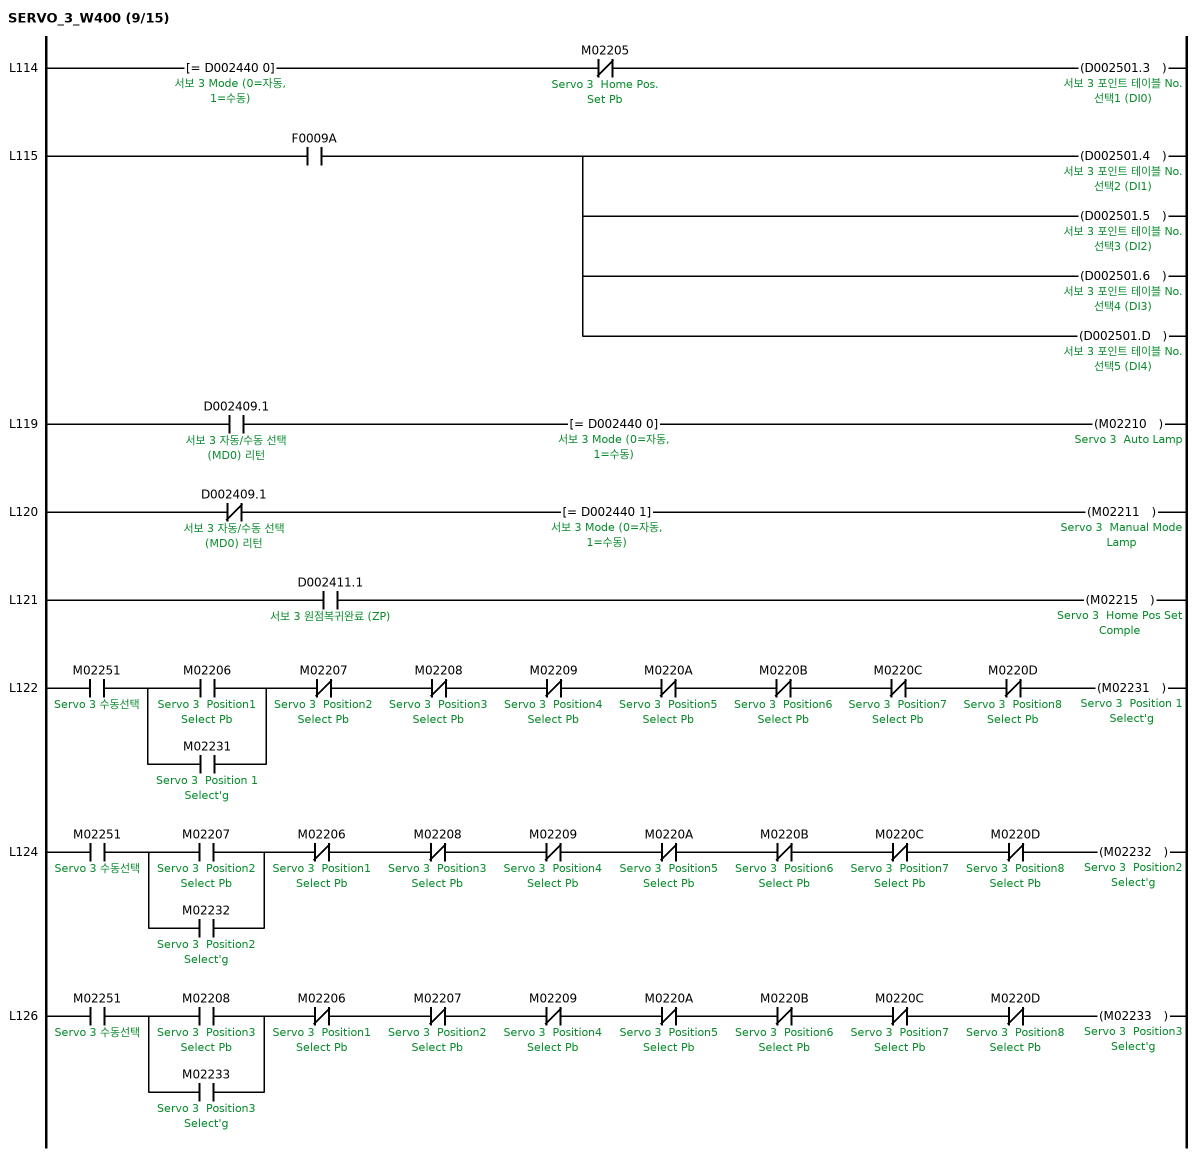
[picture p312: SERVO_3_W400 rungs L114-L126]
; L114
LOAD=     D002440 0	// 서보 3 Mode (0=자동, 1=수동)
AND NOT   M02205	// Servo 3  Home Pos. Set Pb
OUT       D002501.3	// 서보 3 포인트 테이블 No. 선택1 (DI0)
; L115
LOAD      F0009A
OUT       D002501.4	// 서보 3 포인트 테이블 No. 선택2 (DI1)
OUT       D002501.5	// 서보 3 포인트 테이블 No. 선택3 (DI2)
OUT       D002501.6	// 서보 3 포인트 테이블 No. 선택4 (DI3)
OUT       D002501.D	// 서보 3 포인트 테이블 No. 선택5 (DI4)
; L119
LOAD      D002409.1	// 서보 3 자동/수동 선택 (MD0) 리턴
AND=      D002440 0	// 서보 3 Mode (0=자동, 1=수동)
OUT       M02210	// Servo 3  Auto Lamp
; L120
LOAD NOT  D002409.1	// 서보 3 자동/수동 선택 (MD0) 리턴
AND=      D002440 1	// 서보 3 Mode (0=자동, 1=수동)
OUT       M02211	// Servo 3  Manual Mode Lamp
; L121
LOAD      D002411.1	// 서보 3 원점복귀완료 (ZP)
OUT       M02215	// Servo 3  Home Pos Set Comple
; L122
LOAD      M02251	// Servo 3 수동선택
LOAD      M02206	// Servo 3  Position1 Select Pb
OR        M02231	// Servo 3  Position 1 Select'g
AND LOAD
AND NOT   M02207	// Servo 3  Position2 Select Pb
AND NOT   M02208	// Servo 3  Position3 Select Pb
AND NOT   M02209	// Servo 3  Position4 Select Pb
AND NOT   M0220A	// Servo 3  Position5 Select Pb
AND NOT   M0220B	// Servo 3  Position6 Select Pb
AND NOT   M0220C	// Servo 3  Position7 Select Pb
AND NOT   M0220D	// Servo 3  Position8 Select Pb
OUT       M02231	// Servo 3  Position 1 Select'g
; L124
LOAD      M02251	// Servo 3 수동선택
LOAD      M02207	// Servo 3  Position2 Select Pb
OR        M02232	// Servo 3  Position2 Select'g
AND LOAD
AND NOT   M02206	// Servo 3  Position1 Select Pb
AND NOT   M02208	// Servo 3  Position3 Select Pb
AND NOT   M02209	// Servo 3  Position4 Select Pb
AND NOT   M0220A	// Servo 3  Position5 Select Pb
AND NOT   M0220B	// Servo 3  Position6 Select Pb
AND NOT   M0220C	// Servo 3  Position7 Select Pb
AND NOT   M0220D	// Servo 3  Position8 Select Pb
OUT       M02232	// Servo 3  Position2 Select'g
; L126
LOAD      M02251	// Servo 3 수동선택
LOAD      M02208	// Servo 3  Position3 Select Pb
OR        M02233	// Servo 3  Position3 Select'g
AND LOAD
AND NOT   M02206	// Servo 3  Position1 Select Pb
AND NOT   M02207	// Servo 3  Position2 Select Pb
AND NOT   M02209	// Servo 3  Position4 Select Pb
AND NOT   M0220A	// Servo 3  Position5 Select Pb
AND NOT   M0220B	// Servo 3  Position6 Select Pb
AND NOT   M0220C	// Servo 3  Position7 Select Pb
AND NOT   M0220D	// Servo 3  Position8 Select Pb
OUT       M02233	// Servo 3  Position3 Select'g

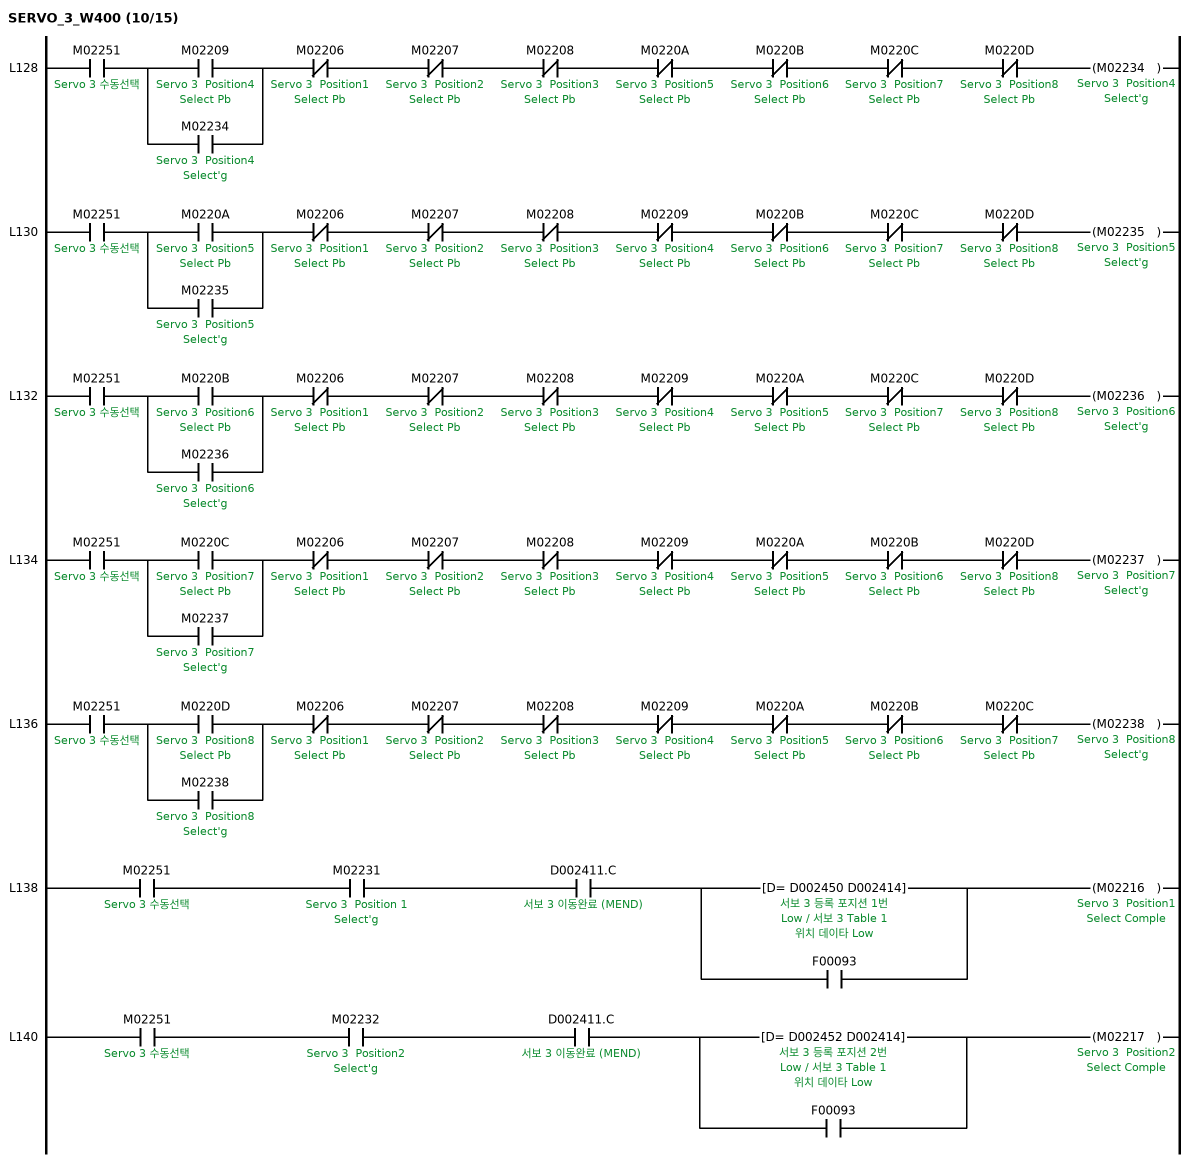
; L128
LOAD      M02251	// Servo 3 수동선택
LOAD      M02209	// Servo 3  Position4 Select Pb
OR        M02234	// Servo 3  Position4 Select'g
AND LOAD
AND NOT   M02206	// Servo 3  Position1 Select Pb
AND NOT   M02207	// Servo 3  Position2 Select Pb
AND NOT   M02208	// Servo 3  Position3 Select Pb
AND NOT   M0220A	// Servo 3  Position5 Select Pb
AND NOT   M0220B	// Servo 3  Position6 Select Pb
AND NOT   M0220C	// Servo 3  Position7 Select Pb
AND NOT   M0220D	// Servo 3  Position8 Select Pb
OUT       M02234	// Servo 3  Position4 Select'g
; L130
LOAD      M02251	// Servo 3 수동선택
LOAD      M0220A	// Servo 3  Position5 Select Pb
OR        M02235	// Servo 3  Position5 Select'g
AND LOAD
AND NOT   M02206	// Servo 3  Position1 Select Pb
AND NOT   M02207	// Servo 3  Position2 Select Pb
AND NOT   M02208	// Servo 3  Position3 Select Pb
AND NOT   M02209	// Servo 3  Position4 Select Pb
AND NOT   M0220B	// Servo 3  Position6 Select Pb
AND NOT   M0220C	// Servo 3  Position7 Select Pb
AND NOT   M0220D	// Servo 3  Position8 Select Pb
OUT       M02235	// Servo 3  Position5 Select'g
; L132
LOAD      M02251	// Servo 3 수동선택
LOAD      M0220B	// Servo 3  Position6 Select Pb
OR        M02236	// Servo 3  Position6 Select'g
AND LOAD
AND NOT   M02206	// Servo 3  Position1 Select Pb
AND NOT   M02207	// Servo 3  Position2 Select Pb
AND NOT   M02208	// Servo 3  Position3 Select Pb
AND NOT   M02209	// Servo 3  Position4 Select Pb
AND NOT   M0220A	// Servo 3  Position5 Select Pb
AND NOT   M0220C	// Servo 3  Position7 Select Pb
AND NOT   M0220D	// Servo 3  Position8 Select Pb
OUT       M02236	// Servo 3  Position6 Select'g
; L134
LOAD      M02251	// Servo 3 수동선택
LOAD      M0220C	// Servo 3  Position7 Select Pb
OR        M02237	// Servo 3  Position7 Select'g
AND LOAD
AND NOT   M02206	// Servo 3  Position1 Select Pb
AND NOT   M02207	// Servo 3  Position2 Select Pb
AND NOT   M02208	// Servo 3  Position3 Select Pb
AND NOT   M02209	// Servo 3  Position4 Select Pb
AND NOT   M0220A	// Servo 3  Position5 Select Pb
AND NOT   M0220B	// Servo 3  Position6 Select Pb
AND NOT   M0220D	// Servo 3  Position8 Select Pb
OUT       M02237	// Servo 3  Position7 Select'g
; L136
LOAD      M02251	// Servo 3 수동선택
LOAD      M0220D	// Servo 3  Position8 Select Pb
OR        M02238	// Servo 3  Position8 Select'g
AND LOAD
AND NOT   M02206	// Servo 3  Position1 Select Pb
AND NOT   M02207	// Servo 3  Position2 Select Pb
AND NOT   M02208	// Servo 3  Position3 Select Pb
AND NOT   M02209	// Servo 3  Position4 Select Pb
AND NOT   M0220A	// Servo 3  Position5 Select Pb
AND NOT   M0220B	// Servo 3  Position6 Select Pb
AND NOT   M0220C	// Servo 3  Position7 Select Pb
OUT       M02238	// Servo 3  Position8 Select'g
; L138
LOAD      M02251	// Servo 3 수동선택
AND       M02231	// Servo 3  Position 1 Select'g
AND       D002411.C	// 서보 3 이동완료 (MEND)
LOADD=    D002450 D002414	// 서보 3 등록 포지션 1번 Low / 서보 3 Table 1 위치 데이타 Low
OR        F00093
AND LOAD
OUT       M02216	// Servo 3  Position1 Select Comple
; L140
LOAD      M02251	// Servo 3 수동선택
AND       M02232	// Servo 3  Position2 Select'g
AND       D002411.C	// 서보 3 이동완료 (MEND)
LOADD=    D002452 D002414	// 서보 3 등록 포지션 2번 Low / 서보 3 Table 1 위치 데이타 Low
OR        F00093
AND LOAD
OUT       M02217	// Servo 3  Position2 Select Comple

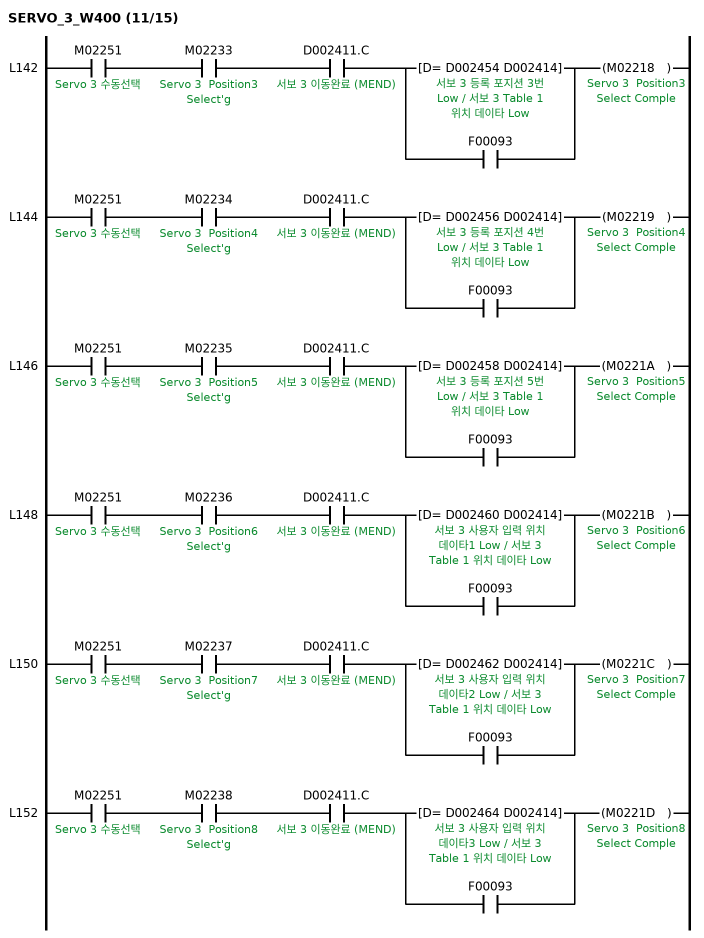
; L142
LOAD      M02251	// Servo 3 수동선택
AND       M02233	// Servo 3  Position3 Select'g
AND       D002411.C	// 서보 3 이동완료 (MEND)
LOADD=    D002454 D002414	// 서보 3 등록 포지션 3번 Low / 서보 3 Table 1 위치 데이타 Low
OR        F00093
AND LOAD
OUT       M02218	// Servo 3  Position3 Select Comple
; L144
LOAD      M02251	// Servo 3 수동선택
AND       M02234	// Servo 3  Position4 Select'g
AND       D002411.C	// 서보 3 이동완료 (MEND)
LOADD=    D002456 D002414	// 서보 3 등록 포지션 4번 Low / 서보 3 Table 1 위치 데이타 Low
OR        F00093
AND LOAD
OUT       M02219	// Servo 3  Position4 Select Comple
; L146
LOAD      M02251	// Servo 3 수동선택
AND       M02235	// Servo 3  Position5 Select'g
AND       D002411.C	// 서보 3 이동완료 (MEND)
LOADD=    D002458 D002414	// 서보 3 등록 포지션 5번 Low / 서보 3 Table 1 위치 데이타 Low
OR        F00093
AND LOAD
OUT       M0221A	// Servo 3  Position5 Select Comple
; L148
LOAD      M02251	// Servo 3 수동선택
AND       M02236	// Servo 3  Position6 Select'g
AND       D002411.C	// 서보 3 이동완료 (MEND)
LOADD=    D002460 D002414	// 서보 3 사용자 입력 위치 데이타1 Low / 서보 3 Table 1 위치 데이타 Low
OR        F00093
AND LOAD
OUT       M0221B	// Servo 3  Position6 Select Comple
; L150
LOAD      M02251	// Servo 3 수동선택
AND       M02237	// Servo 3  Position7 Select'g
AND       D002411.C	// 서보 3 이동완료 (MEND)
LOADD=    D002462 D002414	// 서보 3 사용자 입력 위치 데이타2 Low / 서보 3 Table 1 위치 데이타 Low
OR        F00093
AND LOAD
OUT       M0221C	// Servo 3  Position7 Select Comple
; L152
LOAD      M02251	// Servo 3 수동선택
AND       M02238	// Servo 3  Position8 Select'g
AND       D002411.C	// 서보 3 이동완료 (MEND)
LOADD=    D002464 D002414	// 서보 3 사용자 입력 위치 데이타3 Low / 서보 3 Table 1 위치 데이타 Low
OR        F00093
AND LOAD
OUT       M0221D	// Servo 3  Position8 Select Comple

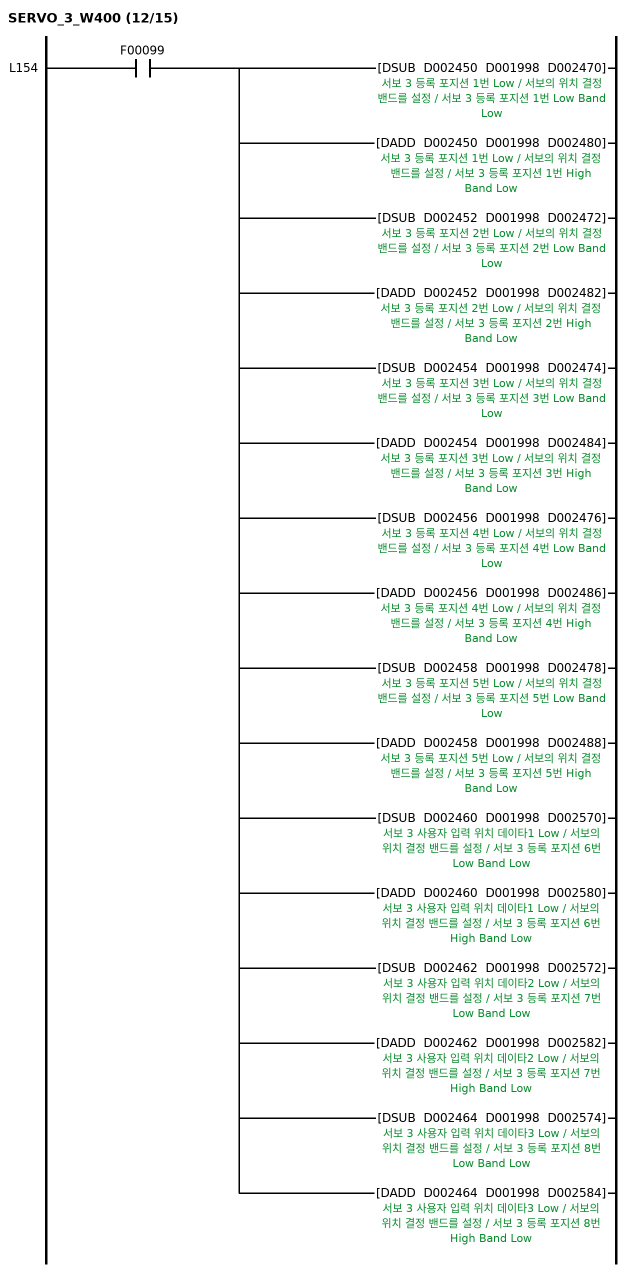
; L154
LOAD      F00099
DSUB      D002450 D001998 D002470	// 서보 3 등록 포지션 1번 Low / 서보의 위치 결정 밴드를 설정 / 서보 3 등록 포지션 1번 Low Band Low
DADD      D002450 D001998 D002480	// 서보 3 등록 포지션 1번 Low / 서보의 위치 결정 밴드를 설정 / 서보 3 등록 포지션 1번 High Band Low
DSUB      D002452 D001998 D002472	// 서보 3 등록 포지션 2번 Low / 서보의 위치 결정 밴드를 설정 / 서보 3 등록 포지션 2번 Low Band Low
DADD      D002452 D001998 D002482	// 서보 3 등록 포지션 2번 Low / 서보의 위치 결정 밴드를 설정 / 서보 3 등록 포지션 2번 High Band Low
DSUB      D002454 D001998 D002474	// 서보 3 등록 포지션 3번 Low / 서보의 위치 결정 밴드를 설정 / 서보 3 등록 포지션 3번 Low Band Low
DADD      D002454 D001998 D002484	// 서보 3 등록 포지션 3번 Low / 서보의 위치 결정 밴드를 설정 / 서보 3 등록 포지션 3번 High Band Low
DSUB      D002456 D001998 D002476	// 서보 3 등록 포지션 4번 Low / 서보의 위치 결정 밴드를 설정 / 서보 3 등록 포지션 4번 Low Band Low
DADD      D002456 D001998 D002486	// 서보 3 등록 포지션 4번 Low / 서보의 위치 결정 밴드를 설정 / 서보 3 등록 포지션 4번 High Band Low
DSUB      D002458 D001998 D002478	// 서보 3 등록 포지션 5번 Low / 서보의 위치 결정 밴드를 설정 / 서보 3 등록 포지션 5번 Low Band Low
DADD      D002458 D001998 D002488	// 서보 3 등록 포지션 5번 Low / 서보의 위치 결정 밴드를 설정 / 서보 3 등록 포지션 5번 High Band Low
DSUB      D002460 D001998 D002570	// 서보 3 사용자 입력 위치 데이타1 Low / 서보의 위치 결정 밴드를 설정 / 서보 3 등록 포지션 6번 Low Band Low
DADD      D002460 D001998 D002580	// 서보 3 사용자 입력 위치 데이타1 Low / 서보의 위치 결정 밴드를 설정 / 서보 3 등록 포지션 6번 High Band Low
DSUB      D002462 D001998 D002572	// 서보 3 사용자 입력 위치 데이타2 Low / 서보의 위치 결정 밴드를 설정 / 서보 3 등록 포지션 7번 Low Band Low
DADD      D002462 D001998 D002582	// 서보 3 사용자 입력 위치 데이타2 Low / 서보의 위치 결정 밴드를 설정 / 서보 3 등록 포지션 7번 High Band Low
DSUB      D002464 D001998 D002574	// 서보 3 사용자 입력 위치 데이타3 Low / 서보의 위치 결정 밴드를 설정 / 서보 3 등록 포지션 8번 Low Band Low
DADD      D002464 D001998 D002584	// 서보 3 사용자 입력 위치 데이타3 Low / 서보의 위치 결정 밴드를 설정 / 서보 3 등록 포지션 8번 High Band Low

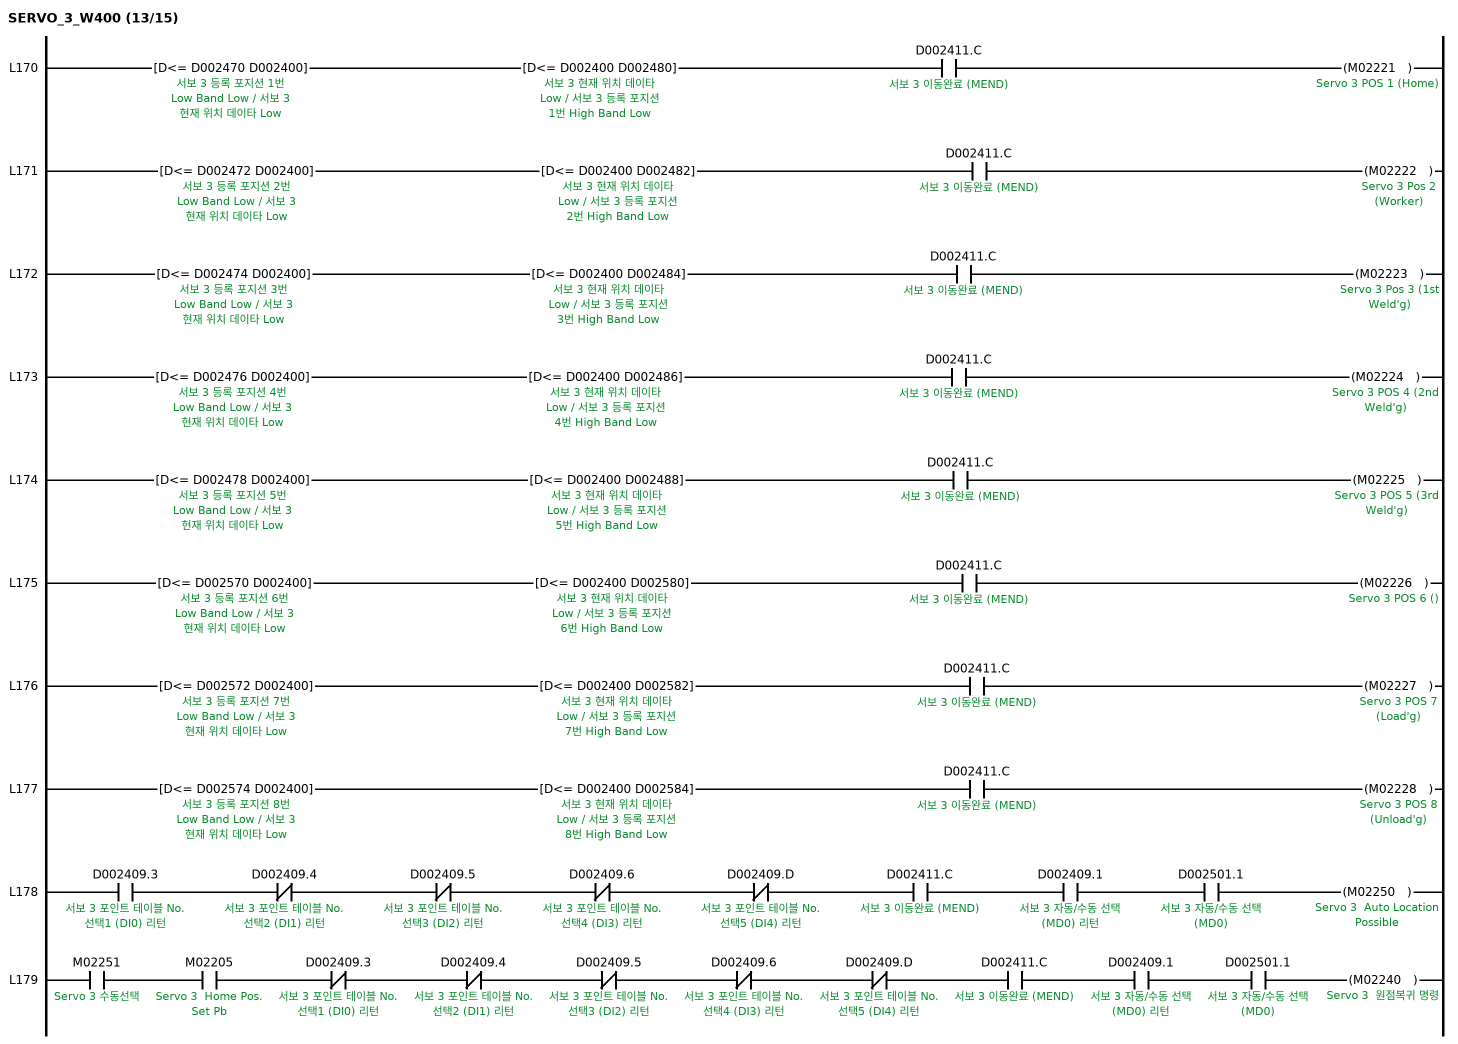
; L170
LOADD<=   D002470 D002400	// 서보 3 등록 포지션 1번 Low Band Low / 서보 3 현재 위치 데이타 Low
ANDD<=    D002400 D002480	// 서보 3 현재 위치 데이타 Low / 서보 3 등록 포지션 1번 High Band Low
AND       D002411.C	// 서보 3 이동완료 (MEND)
OUT       M02221	// Servo 3 POS 1 (Home)
; L171
LOADD<=   D002472 D002400	// 서보 3 등록 포지션 2번 Low Band Low / 서보 3 현재 위치 데이타 Low
ANDD<=    D002400 D002482	// 서보 3 현재 위치 데이타 Low / 서보 3 등록 포지션 2번 High Band Low
AND       D002411.C	// 서보 3 이동완료 (MEND)
OUT       M02222	// Servo 3 Pos 2 (Worker)
; L172
LOADD<=   D002474 D002400	// 서보 3 등록 포지션 3번 Low Band Low / 서보 3 현재 위치 데이타 Low
ANDD<=    D002400 D002484	// 서보 3 현재 위치 데이타 Low / 서보 3 등록 포지션 3번 High Band Low
AND       D002411.C	// 서보 3 이동완료 (MEND)
OUT       M02223	// Servo 3 Pos 3 (1st Weld'g)
; L173
LOADD<=   D002476 D002400	// 서보 3 등록 포지션 4번 Low Band Low / 서보 3 현재 위치 데이타 Low
ANDD<=    D002400 D002486	// 서보 3 현재 위치 데이타 Low / 서보 3 등록 포지션 4번 High Band Low
AND       D002411.C	// 서보 3 이동완료 (MEND)
OUT       M02224	// Servo 3 POS 4 (2nd Weld'g)
; L174
LOADD<=   D002478 D002400	// 서보 3 등록 포지션 5번 Low Band Low / 서보 3 현재 위치 데이타 Low
ANDD<=    D002400 D002488	// 서보 3 현재 위치 데이타 Low / 서보 3 등록 포지션 5번 High Band Low
AND       D002411.C	// 서보 3 이동완료 (MEND)
OUT       M02225	// Servo 3 POS 5 (3rd Weld'g)
; L175
LOADD<=   D002570 D002400	// 서보 3 등록 포지션 6번 Low Band Low / 서보 3 현재 위치 데이타 Low
ANDD<=    D002400 D002580	// 서보 3 현재 위치 데이타 Low / 서보 3 등록 포지션 6번 High Band Low
AND       D002411.C	// 서보 3 이동완료 (MEND)
OUT       M02226	// Servo 3 POS 6 ()
; L176
LOADD<=   D002572 D002400	// 서보 3 등록 포지션 7번 Low Band Low / 서보 3 현재 위치 데이타 Low
ANDD<=    D002400 D002582	// 서보 3 현재 위치 데이타 Low / 서보 3 등록 포지션 7번 High Band Low
AND       D002411.C	// 서보 3 이동완료 (MEND)
OUT       M02227	// Servo 3 POS 7 (Load'g)
; L177
LOADD<=   D002574 D002400	// 서보 3 등록 포지션 8번 Low Band Low / 서보 3 현재 위치 데이타 Low
ANDD<=    D002400 D002584	// 서보 3 현재 위치 데이타 Low / 서보 3 등록 포지션 8번 High Band Low
AND       D002411.C	// 서보 3 이동완료 (MEND)
OUT       M02228	// Servo 3 POS 8 (Unload'g)
; L178
LOAD      D002409.3	// 서보 3 포인트 테이블 No. 선택1 (DI0) 리턴
AND NOT   D002409.4	// 서보 3 포인트 테이블 No. 선택2 (DI1) 리턴
AND NOT   D002409.5	// 서보 3 포인트 테이블 No. 선택3 (DI2) 리턴
AND NOT   D002409.6	// 서보 3 포인트 테이블 No. 선택4 (DI3) 리턴
AND NOT   D002409.D	// 서보 3 포인트 테이블 No. 선택5 (DI4) 리턴
AND       D002411.C	// 서보 3 이동완료 (MEND)
AND       D002409.1	// 서보 3 자동/수동 선택 (MD0) 리턴
AND       D002501.1	// 서보 3 자동/수동 선택 (MD0)
OUT       M02250	// Servo 3  Auto Location Possible
; L179
LOAD      M02251	// Servo 3 수동선택
AND       M02205	// Servo 3  Home Pos. Set Pb
AND NOT   D002409.3	// 서보 3 포인트 테이블 No. 선택1 (DI0) 리턴
AND NOT   D002409.4	// 서보 3 포인트 테이블 No. 선택2 (DI1) 리턴
AND NOT   D002409.5	// 서보 3 포인트 테이블 No. 선택3 (DI2) 리턴
AND NOT   D002409.6	// 서보 3 포인트 테이블 No. 선택4 (DI3) 리턴
AND NOT   D002409.D	// 서보 3 포인트 테이블 No. 선택5 (DI4) 리턴
AND       D002411.C	// 서보 3 이동완료 (MEND)
AND       D002409.1	// 서보 3 자동/수동 선택 (MD0) 리턴
AND       D002501.1	// 서보 3 자동/수동 선택 (MD0)
OUT       M02240	// Servo 3  원점복귀 명령

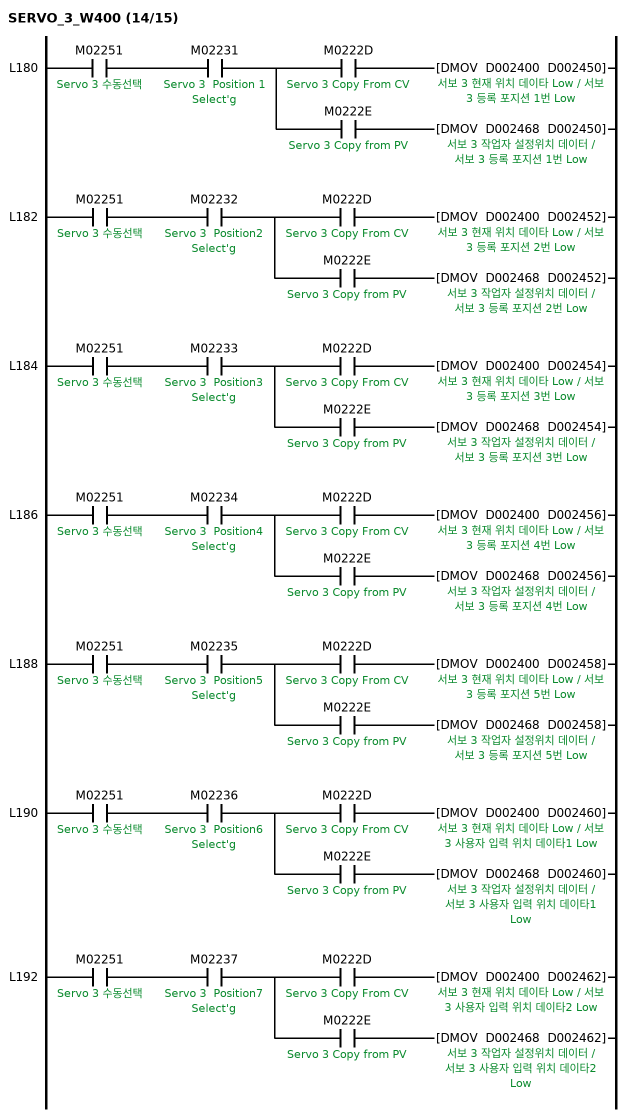
; L180
LOAD      M02251	// Servo 3 수동선택
AND       M02231	// Servo 3  Position 1 Select'g
MPUSH
AND       M0222D	// Servo 3 Copy From CV
DMOV      D002400 D002450	// 서보 3 현재 위치 데이타 Low / 서보 3 등록 포지션 1번 Low
MPOP
AND       M0222E	// Servo 3 Copy from PV
DMOV      D002468 D002450	// 서보 3 작업자 설정위치 데이터 / 서보 3 등록 포지션 1번 Low
; L182
LOAD      M02251	// Servo 3 수동선택
AND       M02232	// Servo 3  Position2 Select'g
MPUSH
AND       M0222D	// Servo 3 Copy From CV
DMOV      D002400 D002452	// 서보 3 현재 위치 데이타 Low / 서보 3 등록 포지션 2번 Low
MPOP
AND       M0222E	// Servo 3 Copy from PV
DMOV      D002468 D002452	// 서보 3 작업자 설정위치 데이터 / 서보 3 등록 포지션 2번 Low
; L184
LOAD      M02251	// Servo 3 수동선택
AND       M02233	// Servo 3  Position3 Select'g
MPUSH
AND       M0222D	// Servo 3 Copy From CV
DMOV      D002400 D002454	// 서보 3 현재 위치 데이타 Low / 서보 3 등록 포지션 3번 Low
MPOP
AND       M0222E	// Servo 3 Copy from PV
DMOV      D002468 D002454	// 서보 3 작업자 설정위치 데이터 / 서보 3 등록 포지션 3번 Low
; L186
LOAD      M02251	// Servo 3 수동선택
AND       M02234	// Servo 3  Position4 Select'g
MPUSH
AND       M0222D	// Servo 3 Copy From CV
DMOV      D002400 D002456	// 서보 3 현재 위치 데이타 Low / 서보 3 등록 포지션 4번 Low
MPOP
AND       M0222E	// Servo 3 Copy from PV
DMOV      D002468 D002456	// 서보 3 작업자 설정위치 데이터 / 서보 3 등록 포지션 4번 Low
; L188
LOAD      M02251	// Servo 3 수동선택
AND       M02235	// Servo 3  Position5 Select'g
MPUSH
AND       M0222D	// Servo 3 Copy From CV
DMOV      D002400 D002458	// 서보 3 현재 위치 데이타 Low / 서보 3 등록 포지션 5번 Low
MPOP
AND       M0222E	// Servo 3 Copy from PV
DMOV      D002468 D002458	// 서보 3 작업자 설정위치 데이터 / 서보 3 등록 포지션 5번 Low
; L190
LOAD      M02251	// Servo 3 수동선택
AND       M02236	// Servo 3  Position6 Select'g
MPUSH
AND       M0222D	// Servo 3 Copy From CV
DMOV      D002400 D002460	// 서보 3 현재 위치 데이타 Low / 서보 3 사용자 입력 위치 데이타1 Low
MPOP
AND       M0222E	// Servo 3 Copy from PV
DMOV      D002468 D002460	// 서보 3 작업자 설정위치 데이터 / 서보 3 사용자 입력 위치 데이타1 Low
; L192
LOAD      M02251	// Servo 3 수동선택
AND       M02237	// Servo 3  Position7 Select'g
MPUSH
AND       M0222D	// Servo 3 Copy From CV
DMOV      D002400 D002462	// 서보 3 현재 위치 데이타 Low / 서보 3 사용자 입력 위치 데이타2 Low
MPOP
AND       M0222E	// Servo 3 Copy from PV
DMOV      D002468 D002462	// 서보 3 작업자 설정위치 데이터 / 서보 3 사용자 입력 위치 데이타2 Low

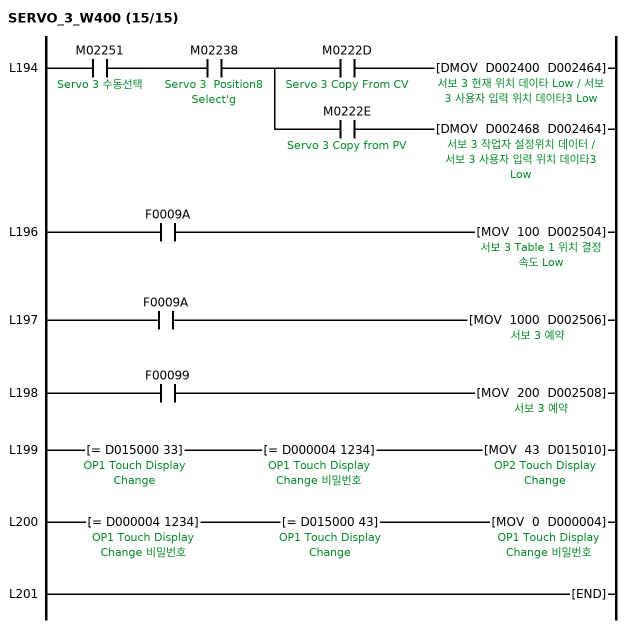
; L194
LOAD      M02251	// Servo 3 수동선택
AND       M02238	// Servo 3  Position8 Select'g
MPUSH
AND       M0222D	// Servo 3 Copy From CV
DMOV      D002400 D002464	// 서보 3 현재 위치 데이타 Low / 서보 3 사용자 입력 위치 데이타3 Low
MPOP
AND       M0222E	// Servo 3 Copy from PV
DMOV      D002468 D002464	// 서보 3 작업자 설정위치 데이터 / 서보 3 사용자 입력 위치 데이타3 Low
; L196
LOAD      F0009A
MOV       100 D002504	// 서보 3 Table 1 위치 결정 속도 Low
; L197
LOAD      F0009A
MOV       1000 D002506	// 서보 3 예약
; L198
LOAD      F00099
MOV       200 D002508	// 서보 3 예약
; L199
LOAD=     D015000 33	// OP1 Touch Display Change
AND=      D000004 1234	// OP1 Touch Display Change 비밀번호
MOV       43 D015010	// OP2 Touch Display Change
; L200
LOAD=     D000004 1234	// OP1 Touch Display Change 비밀번호
AND=      D015000 43	// OP1 Touch Display Change
MOV       0 D000004	// OP1 Touch Display Change 비밀번호
; L201
END

PROGRAM Robot_01_ARC (task: 스캔 프로그램)

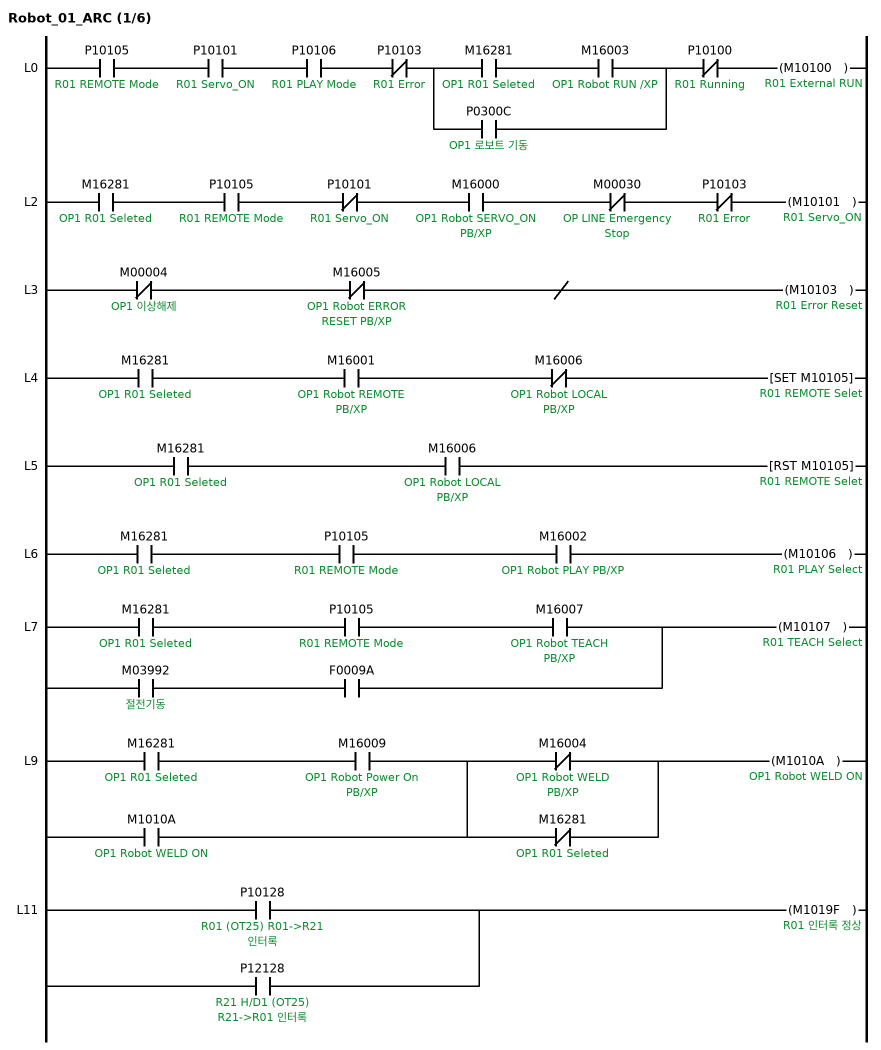
; L0
LOAD      P10105	// R01 REMOTE Mode
AND       P10101	// R01 Servo_ON
AND       P10106	// R01 PLAY Mode
AND NOT   P10103	// R01 Error
LOAD      M16281	// OP1 R01 Seleted
AND       M16003	// OP1 Robot RUN /XP
OR        P0300C	// OP1 로보트 기동
AND LOAD
AND NOT   P10100	// R01 Running
OUT       M10100	// R01 External RUN
; L2
LOAD      M16281	// OP1 R01 Seleted
AND       P10105	// R01 REMOTE Mode
AND NOT   P10101	// R01 Servo_ON
AND       M16000	// OP1 Robot SERVO_ON PB/XP
AND NOT   M00030	// OP LINE Emergency Stop
AND NOT   P10103	// R01 Error
OUT       M10101	// R01 Servo_ON
; L3
LOAD NOT  M00004	// OP1 이상해제
AND NOT   M16005	// OP1 Robot ERROR RESET PB/XP
NOT
OUT       M10103	// R01 Error Reset
; L4
LOAD      M16281	// OP1 R01 Seleted
AND       M16001	// OP1 Robot REMOTE PB/XP
AND NOT   M16006	// OP1 Robot LOCAL PB/XP
SET       M10105	// R01 REMOTE Selet
; L5
LOAD      M16281	// OP1 R01 Seleted
AND       M16006	// OP1 Robot LOCAL PB/XP
RST       M10105	// R01 REMOTE Selet
; L6
LOAD      M16281	// OP1 R01 Seleted
AND       P10105	// R01 REMOTE Mode
AND       M16002	// OP1 Robot PLAY PB/XP
OUT       M10106	// R01 PLAY Select
; L7
LOAD      M16281	// OP1 R01 Seleted
AND       P10105	// R01 REMOTE Mode
AND       M16007	// OP1 Robot TEACH PB/XP
LOAD      M03992	// 절전기동
AND       F0009A
OR LOAD
OUT       M10107	// R01 TEACH Select
; L9
LOAD      M16281	// OP1 R01 Seleted
AND       M16009	// OP1 Robot Power On PB/XP
OR        M1010A	// OP1 Robot WELD ON
LOAD NOT  M16004	// OP1 Robot WELD PB/XP
OR NOT    M16281	// OP1 R01 Seleted
AND LOAD
OUT       M1010A	// OP1 Robot WELD ON
; L11
LOAD      P10128	// R01 (OT25) R01->R21 인터록
OR        P12128	// R21 H/D1 (OT25) R21->R01 인터록
OUT       M1019F	// R01 인터록 정상

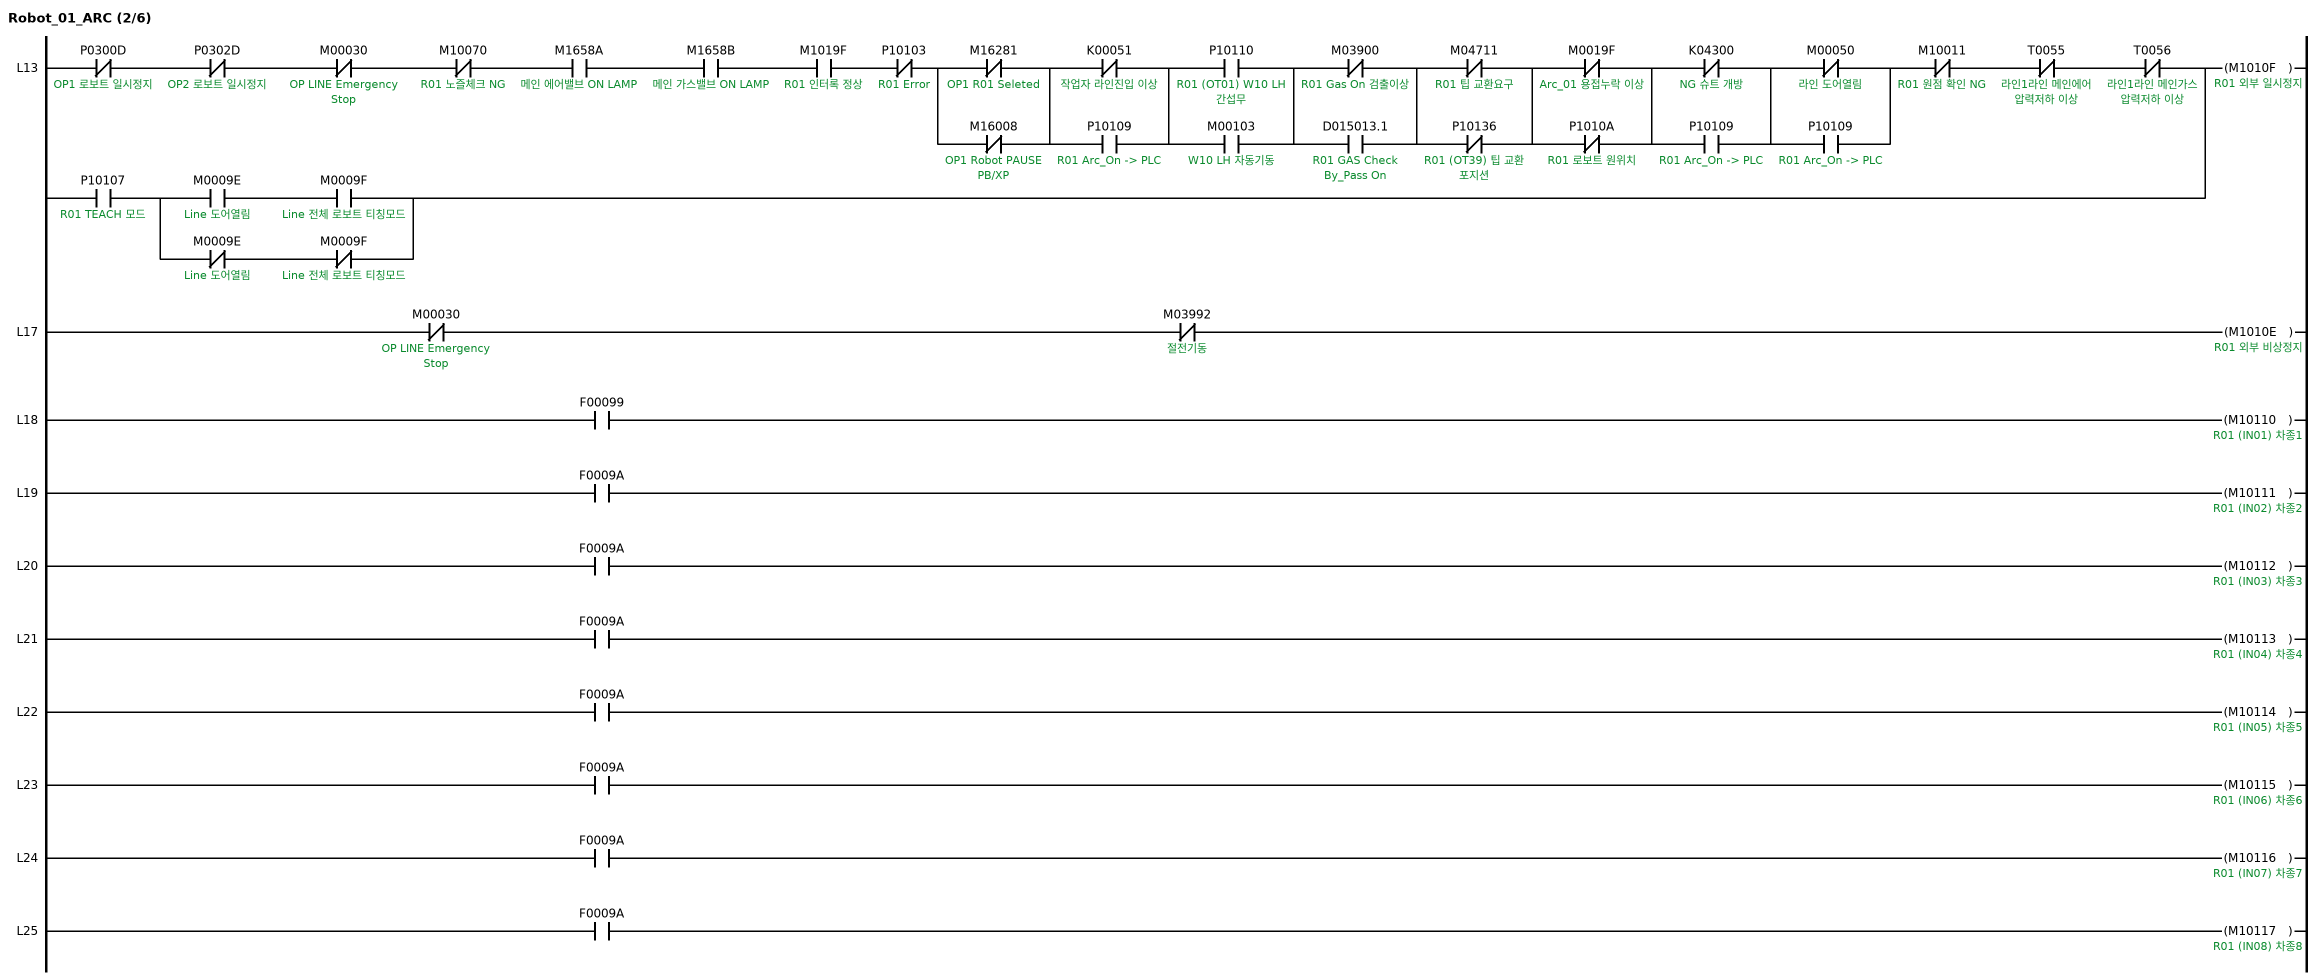
; L13
LOAD NOT  P0300D	// OP1 로보트 일시정지
AND NOT   P0302D	// OP2 로보트 일시정지
AND NOT   M00030	// OP LINE Emergency Stop
AND NOT   M10070	// R01 노즐체크 NG
AND       M1658A	// 메인 에어밸브 ON LAMP
AND       M1658B	// 메인 가스밸브 ON LAMP
AND       M1019F	// R01 인터록 정상
AND NOT   P10103	// R01 Error
LOAD NOT  M16281	// OP1 R01 Seleted
OR NOT    M16008	// OP1 Robot PAUSE PB/XP
AND LOAD
LOAD NOT  K00051	//  작업자 라인진입 이상
OR        P10109	// R01 Arc_On -> PLC
AND LOAD
LOAD      P10110	// R01 (OT01) W10 LH 간섭무
OR        M00103	// W10 LH 자동기동
AND LOAD
LOAD NOT  M03900	// R01 Gas On 검출이상
OR        D015013.1	// R01 GAS Check By_Pass On
AND LOAD
LOAD NOT  M04711	// R01 팁 교환요구
OR NOT    P10136	// R01 (OT39) 팁 교환 포지션
AND LOAD
LOAD NOT  M0019F	// Arc_01 용접누락 이상
OR NOT    P1010A	// R01 로보트 원위치
AND LOAD
LOAD NOT  K04300	// NG 슈트 개방
OR        P10109	// R01 Arc_On -> PLC
AND LOAD
LOAD NOT  M00050	// 라인 도어열림
OR        P10109	// R01 Arc_On -> PLC
AND LOAD
AND NOT   M10011	// R01 원점 확인 NG
AND NOT   T0055	// 라인1라인 메인에어 압력저하 이상
AND NOT   T0056	// 라인1라인 메인가스 압력저하 이상
LOAD      P10107	// R01 TEACH 모드
LOAD      M0009E	// Line 도어열림
AND       M0009F	// Line 전체 로보트 티칭모드
LOAD NOT  M0009E	// Line 도어열림
AND NOT   M0009F	// Line 전체 로보트 티칭모드
OR LOAD
AND LOAD
OR LOAD
OUT       M1010F	// R01 외부 일시정지
; L17
LOAD NOT  M00030	// OP LINE Emergency Stop
AND NOT   M03992	// 절전기동
OUT       M1010E	// R01 외부 비상정지 
; L18
LOAD      F00099
OUT       M10110	// R01 (IN01) 차종1
; L19
LOAD      F0009A
OUT       M10111	// R01 (IN02) 차종2
; L20
LOAD      F0009A
OUT       M10112	// R01 (IN03) 차종3
; L21
LOAD      F0009A
OUT       M10113	// R01 (IN04) 차종4
; L22
LOAD      F0009A
OUT       M10114	// R01 (IN05) 차종5
; L23
LOAD      F0009A
OUT       M10115	// R01 (IN06) 차종6
; L24
LOAD      F0009A
OUT       M10116	// R01 (IN07) 차종7
; L25
LOAD      F0009A
OUT       M10117	// R01 (IN08) 차종8

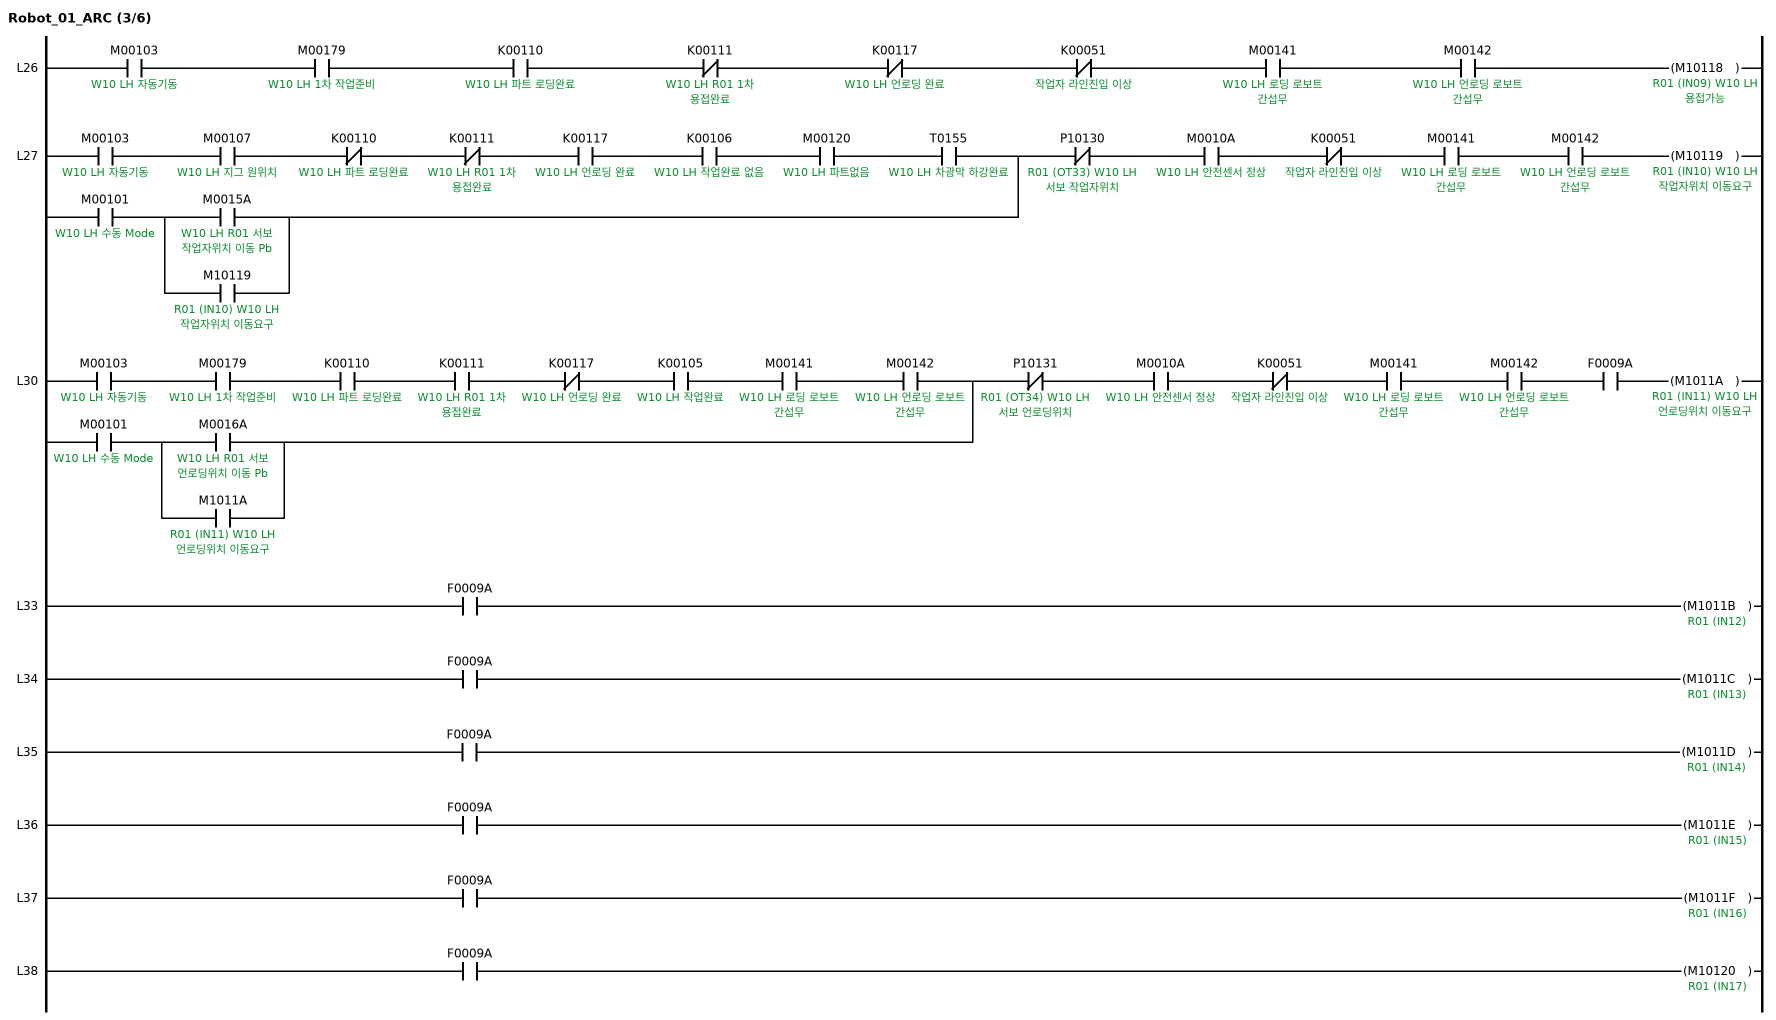
; L26
LOAD      M00103	// W10 LH 자동기동
AND       M00179	// W10 LH 1차 작업준비
AND       K00110	// W10 LH 파트 로딩완료
AND NOT   K00111	// W10 LH R01 1차 용접완료
AND NOT   K00117	// W10 LH 언로딩 완료
AND NOT   K00051	//  작업자 라인진입 이상
AND       M00141	// W10 LH 로딩 로보트 간섭무
AND       M00142	// W10 LH 언로딩 로보트 간섭무
OUT       M10118	// R01 (IN09) W10 LH 용접가능
; L27
LOAD      M00103	// W10 LH 자동기동
AND       M00107	// W10 LH 지그 원위치
AND NOT   K00110	// W10 LH 파트 로딩완료
AND NOT   K00111	// W10 LH R01 1차 용접완료
AND       K00117	// W10 LH 언로딩 완료
AND       K00106	// W10 LH 작업완료 없음
AND       M00120	// W10 LH 파트없음
AND       T0155	// W10 LH 차광막 하강완료
LOAD      M00101	// W10 LH 수동 Mode
LOAD      M0015A	// W10 LH R01 서보 작업자위치 이동 Pb
OR        M10119	// R01 (IN10) W10 LH 작업자위치 이동요구
AND LOAD
OR LOAD
AND NOT   P10130	// R01 (OT33) W10 LH 서보 작업자위치
AND       M0010A	// W10 LH 안전센서 정상
AND NOT   K00051	//  작업자 라인진입 이상
AND       M00141	// W10 LH 로딩 로보트 간섭무
AND       M00142	// W10 LH 언로딩 로보트 간섭무
OUT       M10119	// R01 (IN10) W10 LH 작업자위치 이동요구
; L30
LOAD      M00103	// W10 LH 자동기동
AND       M00179	// W10 LH 1차 작업준비
AND       K00110	// W10 LH 파트 로딩완료
AND       K00111	// W10 LH R01 1차 용접완료
AND NOT   K00117	// W10 LH 언로딩 완료
AND       K00105	// W10 LH 작업완료
AND       M00141	// W10 LH 로딩 로보트 간섭무
AND       M00142	// W10 LH 언로딩 로보트 간섭무
LOAD      M00101	// W10 LH 수동 Mode
LOAD      M0016A	// W10 LH R01 서보 언로딩위치 이동 Pb
OR        M1011A	// R01 (IN11) W10 LH 언로딩위치 이동요구
AND LOAD
OR LOAD
AND NOT   P10131	// R01 (OT34) W10 LH 서보 언로딩위치
AND       M0010A	// W10 LH 안전센서 정상
AND NOT   K00051	//  작업자 라인진입 이상
AND       M00141	// W10 LH 로딩 로보트 간섭무
AND       M00142	// W10 LH 언로딩 로보트 간섭무
AND       F0009A
OUT       M1011A	// R01 (IN11) W10 LH 언로딩위치 이동요구
; L33
LOAD      F0009A
OUT       M1011B	// R01 (IN12)
; L34
LOAD      F0009A
OUT       M1011C	// R01 (IN13)
; L35
LOAD      F0009A
OUT       M1011D	// R01 (IN14)
; L36
LOAD      F0009A
OUT       M1011E	// R01 (IN15)
; L37
LOAD      F0009A
OUT       M1011F	// R01 (IN16)
; L38
LOAD      F0009A
OUT       M10120	// R01 (IN17)

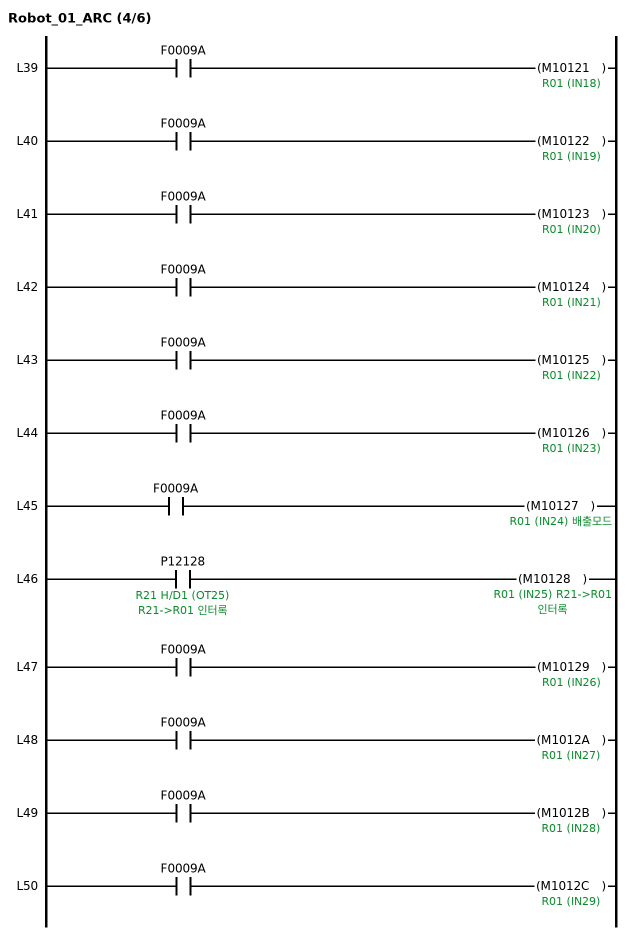
; L39
LOAD      F0009A
OUT       M10121	// R01 (IN18)
; L40
LOAD      F0009A
OUT       M10122	// R01 (IN19)
; L41
LOAD      F0009A
OUT       M10123	// R01 (IN20)
; L42
LOAD      F0009A
OUT       M10124	// R01 (IN21)
; L43
LOAD      F0009A
OUT       M10125	// R01 (IN22)
; L44
LOAD      F0009A
OUT       M10126	// R01 (IN23)
; L45
LOAD      F0009A
OUT       M10127	// R01 (IN24) 배출모드
; L46
LOAD      P12128	// R21 H/D1 (OT25) R21->R01 인터록
OUT       M10128	// R01 (IN25) R21->R01 인터록
; L47
LOAD      F0009A
OUT       M10129	// R01 (IN26)
; L48
LOAD      F0009A
OUT       M1012A	// R01 (IN27)
; L49
LOAD      F0009A
OUT       M1012B	// R01 (IN28)
; L50
LOAD      F0009A
OUT       M1012C	// R01 (IN29)

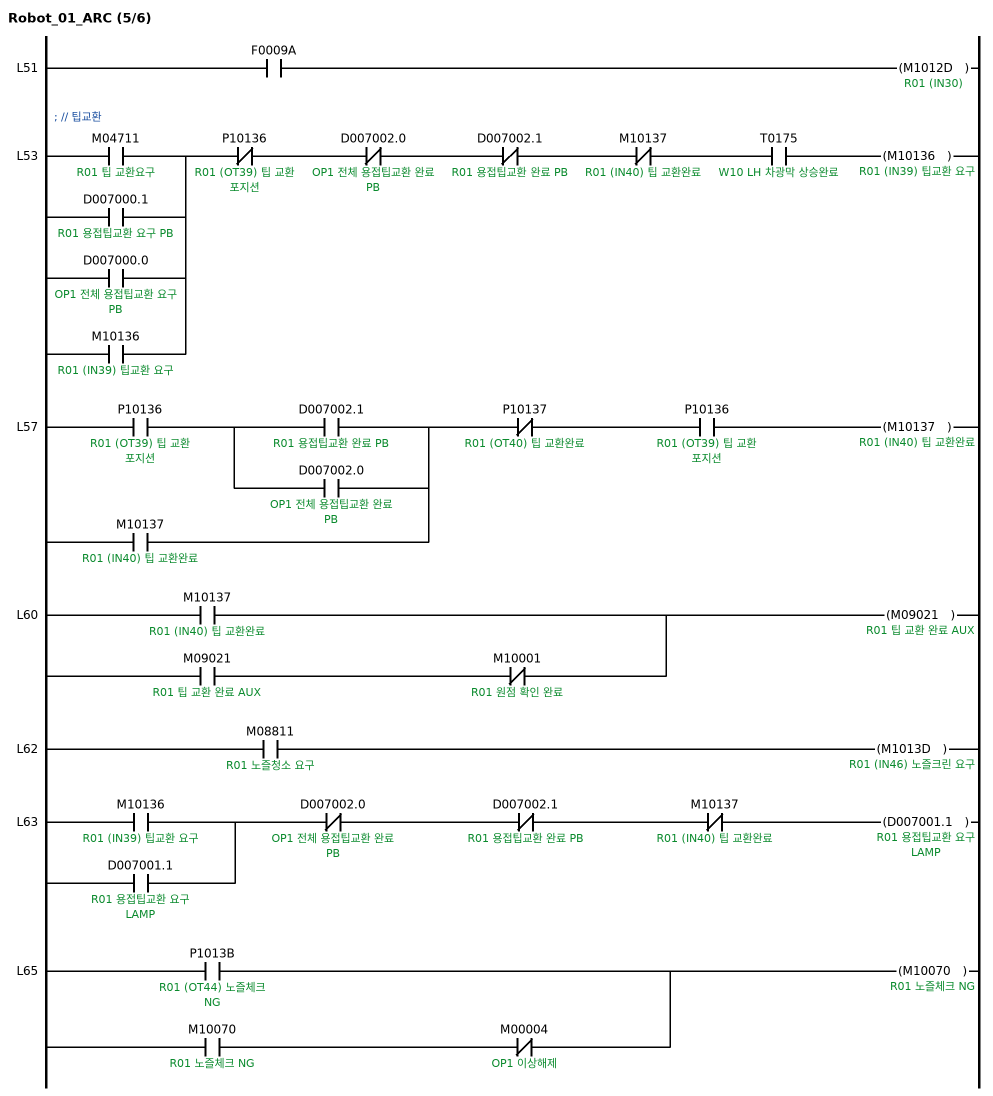
; L51
LOAD      F0009A
OUT       M1012D	// R01 (IN30)
//  // 팁교환
; L53
LOAD      M04711	// R01 팁 교환요구
OR        D007000.1	// R01 용접팁교환 요구 PB
OR        D007000.0	// OP1 전체 용접팁교환 요구 PB
OR        M10136	// R01 (IN39) 팁교환 요구
AND NOT   P10136	// R01 (OT39) 팁 교환 포지션
AND NOT   D007002.0	// OP1 전체 용접팁교환 완료 PB
AND NOT   D007002.1	// R01 용접팁교환 완료 PB
AND NOT   M10137	// R01 (IN40) 팁 교환완료
AND       T0175	// W10 LH 차광막 상승완료
OUT       M10136	// R01 (IN39) 팁교환 요구
; L57
LOAD      P10136	// R01 (OT39) 팁 교환 포지션
LOAD      D007002.1	// R01 용접팁교환 완료 PB
OR        D007002.0	// OP1 전체 용접팁교환 완료 PB
AND LOAD
OR        M10137	// R01 (IN40) 팁 교환완료
AND NOT   P10137	// R01 (OT40) 팁 교환완료
AND       P10136	// R01 (OT39) 팁 교환 포지션
OUT       M10137	// R01 (IN40) 팁 교환완료
; L60
LOAD      M10137	// R01 (IN40) 팁 교환완료
LOAD      M09021	// R01 팁 교환 완료 AUX
AND NOT   M10001	// R01 원점 확인 완료
OR LOAD
OUT       M09021	// R01 팁 교환 완료 AUX
; L62
LOAD      M08811	// R01 노즐청소 요구
OUT       M1013D	// R01 (IN46) 노즐크린 요구
; L63
LOAD      M10136	// R01 (IN39) 팁교환 요구
OR        D007001.1	// R01 용접팁교환 요구 LAMP
AND NOT   D007002.0	// OP1 전체 용접팁교환 완료 PB
AND NOT   D007002.1	// R01 용접팁교환 완료 PB
AND NOT   M10137	// R01 (IN40) 팁 교환완료
OUT       D007001.1	// R01 용접팁교환 요구 LAMP
; L65
LOAD      P1013B	// R01 (OT44) 노즐체크 NG
LOAD      M10070	// R01 노즐체크 NG
AND NOT   M00004	// OP1 이상해제
OR LOAD
OUT       M10070	// R01 노즐체크 NG

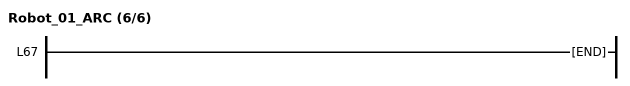
; L67
END

PROGRAM Robot_02_ARC (task: 스캔 프로그램)

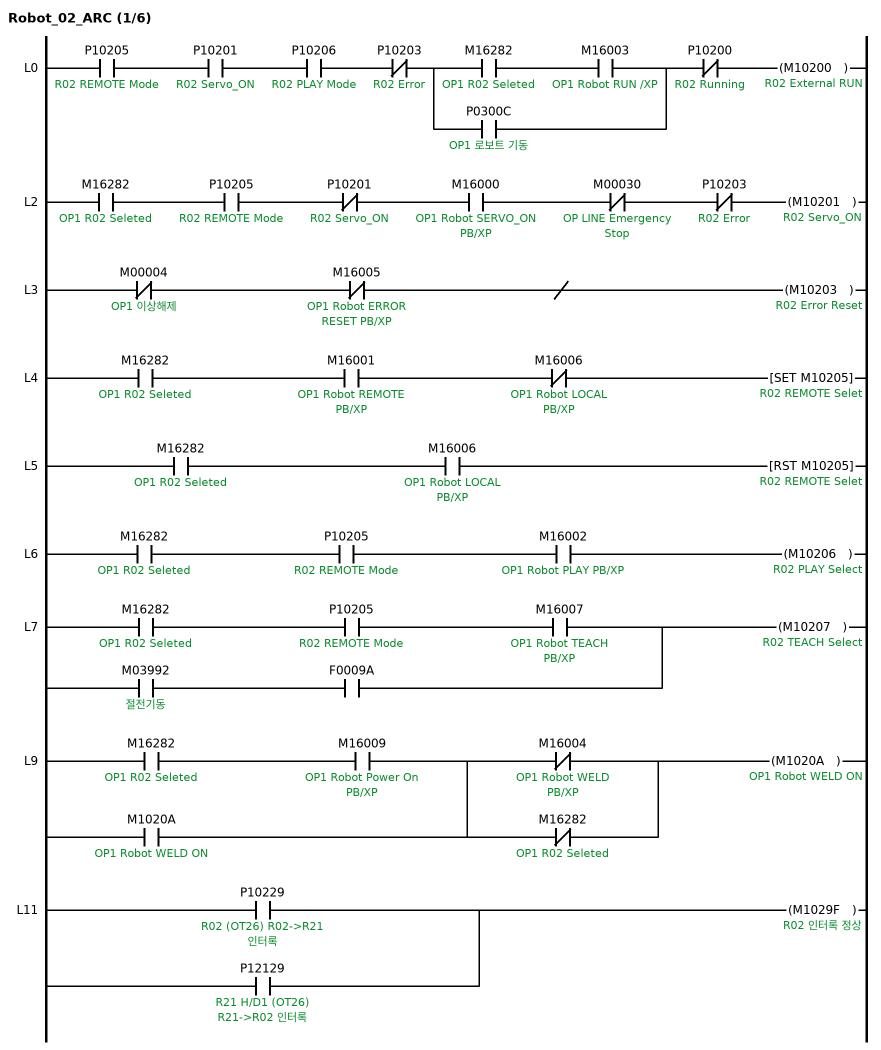
; L0
LOAD      P10205	// R02 REMOTE Mode
AND       P10201	// R02 Servo_ON
AND       P10206	// R02 PLAY Mode
AND NOT   P10203	// R02 Error
LOAD      M16282	// OP1 R02 Seleted
AND       M16003	// OP1 Robot RUN /XP
OR        P0300C	// OP1 로보트 기동
AND LOAD
AND NOT   P10200	// R02 Running
OUT       M10200	// R02 External RUN
; L2
LOAD      M16282	// OP1 R02 Seleted
AND       P10205	// R02 REMOTE Mode
AND NOT   P10201	// R02 Servo_ON
AND       M16000	// OP1 Robot SERVO_ON PB/XP
AND NOT   M00030	// OP LINE Emergency Stop
AND NOT   P10203	// R02 Error
OUT       M10201	// R02 Servo_ON
; L3
LOAD NOT  M00004	// OP1 이상해제
AND NOT   M16005	// OP1 Robot ERROR RESET PB/XP
NOT
OUT       M10203	// R02 Error Reset
; L4
LOAD      M16282	// OP1 R02 Seleted
AND       M16001	// OP1 Robot REMOTE PB/XP
AND NOT   M16006	// OP1 Robot LOCAL PB/XP
SET       M10205	// R02 REMOTE Selet
; L5
LOAD      M16282	// OP1 R02 Seleted
AND       M16006	// OP1 Robot LOCAL PB/XP
RST       M10205	// R02 REMOTE Selet
; L6
LOAD      M16282	// OP1 R02 Seleted
AND       P10205	// R02 REMOTE Mode
AND       M16002	// OP1 Robot PLAY PB/XP
OUT       M10206	// R02 PLAY Select
; L7
LOAD      M16282	// OP1 R02 Seleted
AND       P10205	// R02 REMOTE Mode
AND       M16007	// OP1 Robot TEACH PB/XP
LOAD      M03992	// 절전기동
AND       F0009A
OR LOAD
OUT       M10207	// R02 TEACH Select
; L9
LOAD      M16282	// OP1 R02 Seleted
AND       M16009	// OP1 Robot Power On PB/XP
OR        M1020A	// OP1 Robot WELD ON
LOAD NOT  M16004	// OP1 Robot WELD PB/XP
OR NOT    M16282	// OP1 R02 Seleted
AND LOAD
OUT       M1020A	// OP1 Robot WELD ON
; L11
LOAD      P10229	// R02 (OT26) R02->R21 인터록
OR        P12129	// R21 H/D1 (OT26) R21->R02 인터록
OUT       M1029F	// R02 인터록 정상

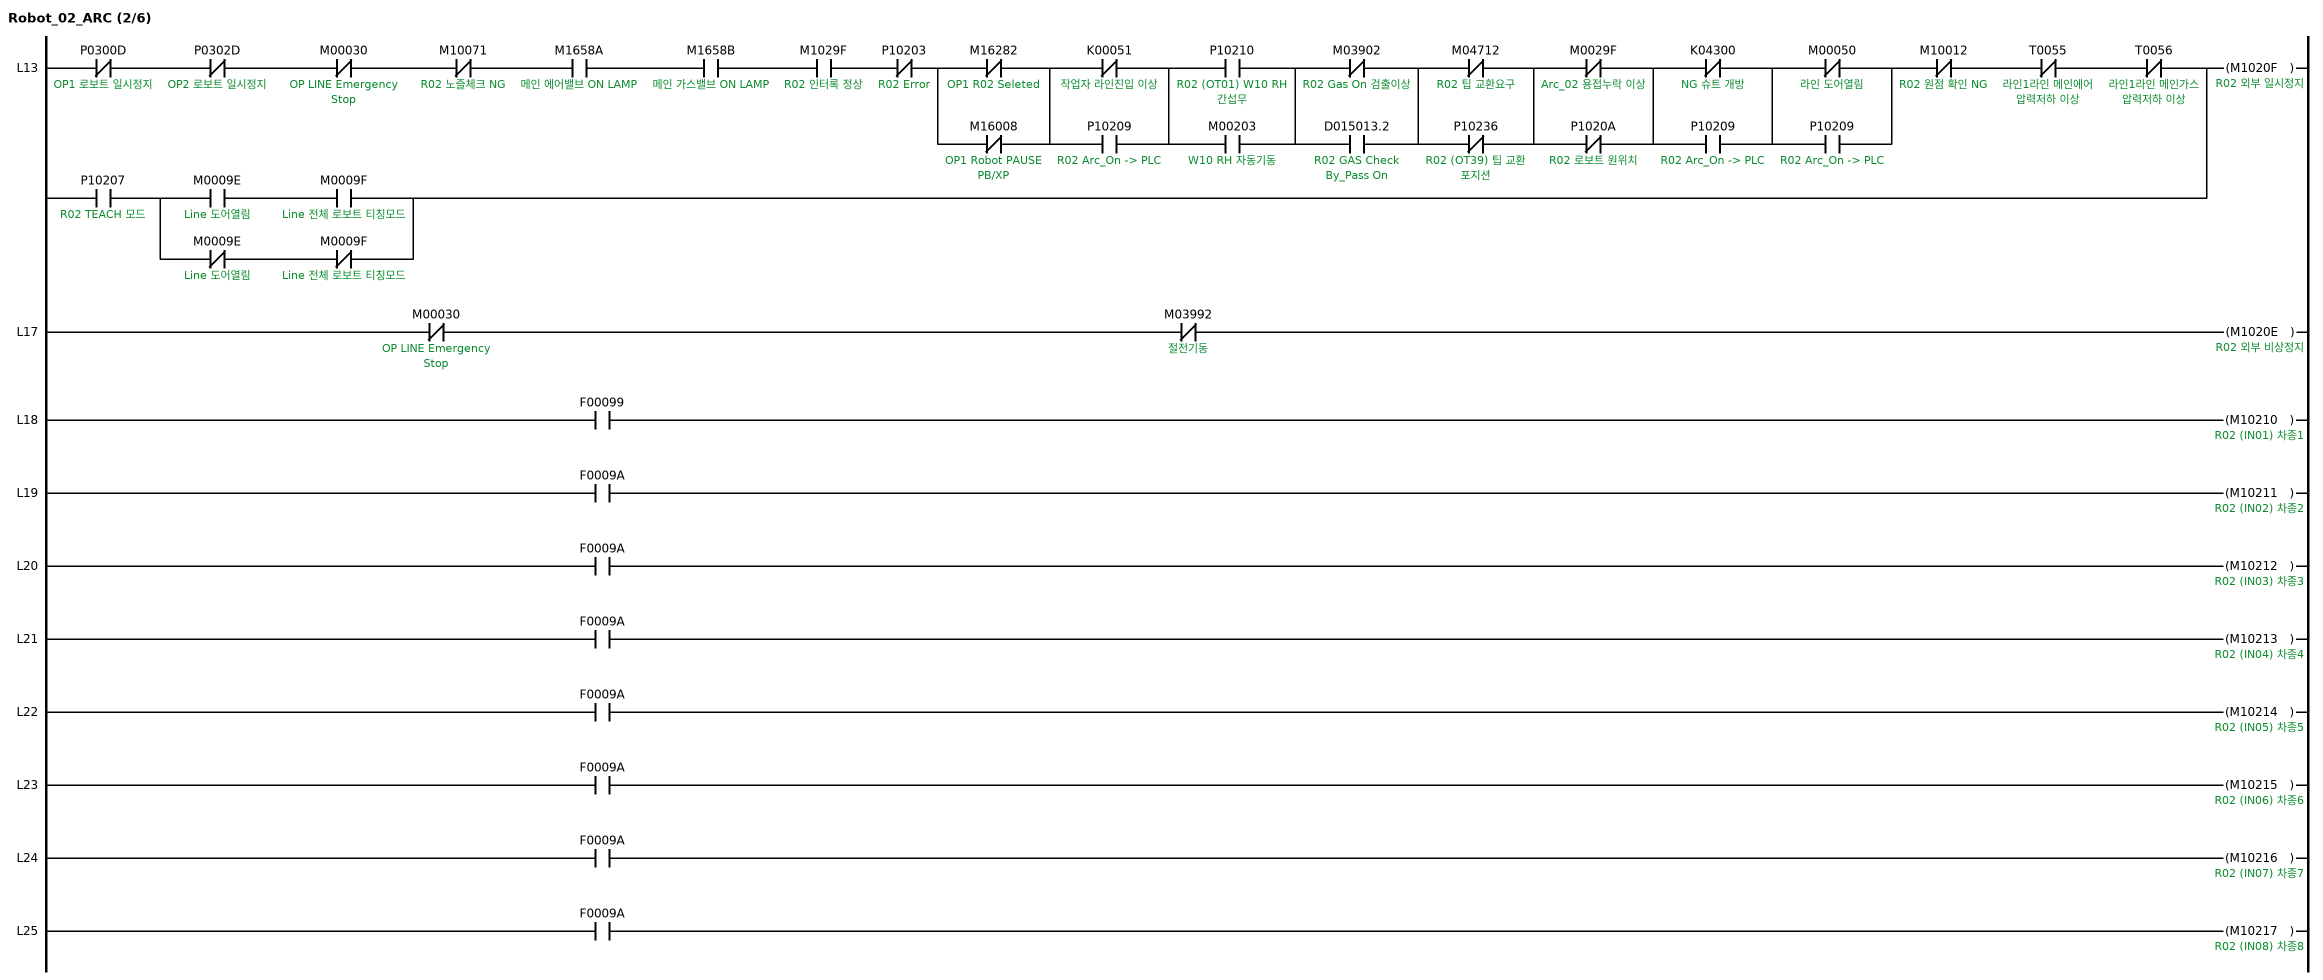
; L13
LOAD NOT  P0300D	// OP1 로보트 일시정지
AND NOT   P0302D	// OP2 로보트 일시정지
AND NOT   M00030	// OP LINE Emergency Stop
AND NOT   M10071	// R02 노즐체크 NG
AND       M1658A	// 메인 에어밸브 ON LAMP
AND       M1658B	// 메인 가스밸브 ON LAMP
AND       M1029F	// R02 인터록 정상
AND NOT   P10203	// R02 Error
LOAD NOT  M16282	// OP1 R02 Seleted
OR NOT    M16008	// OP1 Robot PAUSE PB/XP
AND LOAD
LOAD NOT  K00051	//  작업자 라인진입 이상
OR        P10209	// R02 Arc_On -> PLC
AND LOAD
LOAD      P10210	// R02 (OT01) W10 RH 간섭무
OR        M00203	// W10 RH 자동기동
AND LOAD
LOAD NOT  M03902	// R02 Gas On 검출이상
OR        D015013.2	// R02 GAS Check By_Pass On
AND LOAD
LOAD NOT  M04712	// R02 팁 교환요구
OR NOT    P10236	// R02 (OT39) 팁 교환 포지션
AND LOAD
LOAD NOT  M0029F	// Arc_02 용접누락 이상
OR NOT    P1020A	// R02 로보트 원위치
AND LOAD
LOAD NOT  K04300	// NG 슈트 개방
OR        P10209	// R02 Arc_On -> PLC
AND LOAD
LOAD NOT  M00050	// 라인 도어열림
OR        P10209	// R02 Arc_On -> PLC
AND LOAD
AND NOT   M10012	// R02 원점 확인 NG
AND NOT   T0055	// 라인1라인 메인에어 압력저하 이상
AND NOT   T0056	// 라인1라인 메인가스 압력저하 이상
LOAD      P10207	// R02 TEACH 모드
LOAD      M0009E	// Line 도어열림
AND       M0009F	// Line 전체 로보트 티칭모드
LOAD NOT  M0009E	// Line 도어열림
AND NOT   M0009F	// Line 전체 로보트 티칭모드
OR LOAD
AND LOAD
OR LOAD
OUT       M1020F	// R02 외부 일시정지
; L17
LOAD NOT  M00030	// OP LINE Emergency Stop
AND NOT   M03992	// 절전기동
OUT       M1020E	// R02 외부 비상정지 
; L18
LOAD      F00099
OUT       M10210	// R02 (IN01) 차종1
; L19
LOAD      F0009A
OUT       M10211	// R02 (IN02) 차종2
; L20
LOAD      F0009A
OUT       M10212	// R02 (IN03) 차종3
; L21
LOAD      F0009A
OUT       M10213	// R02 (IN04) 차종4
; L22
LOAD      F0009A
OUT       M10214	// R02 (IN05) 차종5
; L23
LOAD      F0009A
OUT       M10215	// R02 (IN06) 차종6
; L24
LOAD      F0009A
OUT       M10216	// R02 (IN07) 차종7
; L25
LOAD      F0009A
OUT       M10217	// R02 (IN08) 차종8

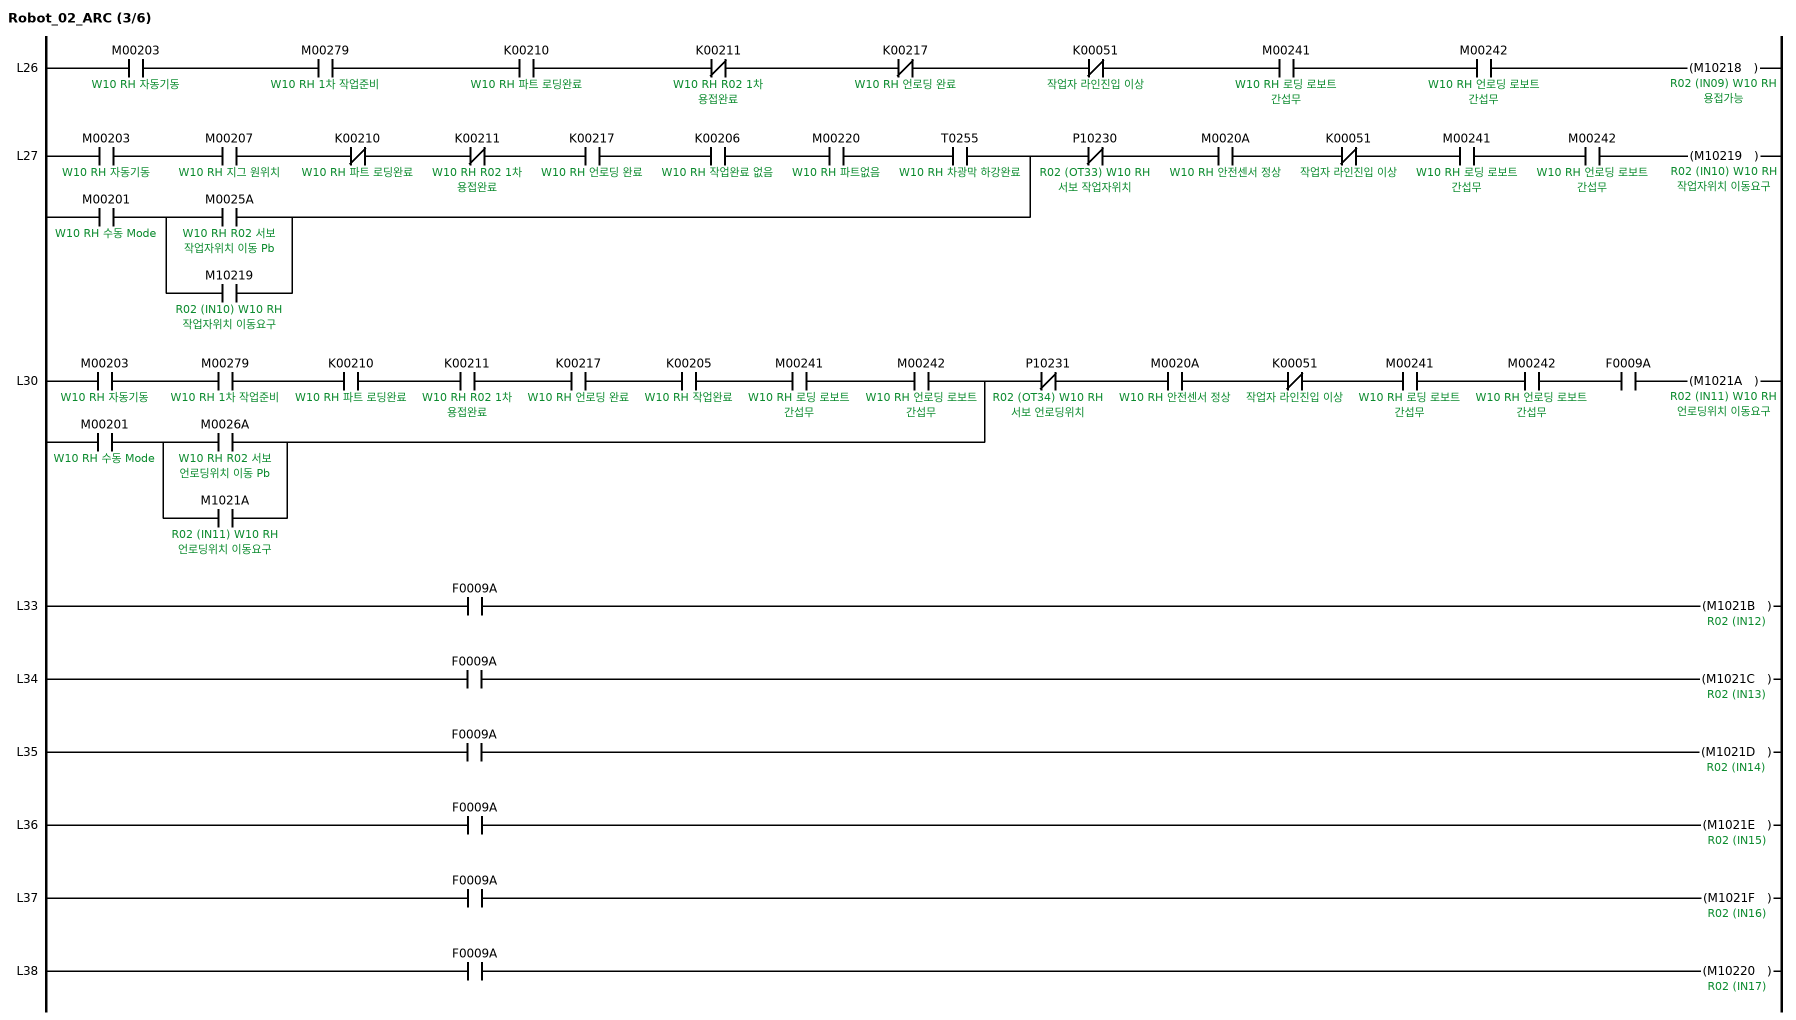
; L26
LOAD      M00203	// W10 RH 자동기동
AND       M00279	// W10 RH 1차 작업준비
AND       K00210	// W10 RH 파트 로딩완료
AND NOT   K00211	// W10 RH R02 1차 용접완료
AND NOT   K00217	// W10 RH 언로딩 완료
AND NOT   K00051	//  작업자 라인진입 이상
AND       M00241	// W10 RH 로딩 로보트 간섭무
AND       M00242	// W10 RH 언로딩 로보트 간섭무
OUT       M10218	// R02 (IN09) W10 RH 용접가능
; L27
LOAD      M00203	// W10 RH 자동기동
AND       M00207	// W10 RH 지그 원위치
AND NOT   K00210	// W10 RH 파트 로딩완료
AND NOT   K00211	// W10 RH R02 1차 용접완료
AND       K00217	// W10 RH 언로딩 완료
AND       K00206	// W10 RH 작업완료 없음
AND       M00220	// W10 RH 파트없음
AND       T0255	// W10 RH 차광막 하강완료
LOAD      M00201	// W10 RH 수동 Mode
LOAD      M0025A	// W10 RH R02 서보 작업자위치 이동 Pb
OR        M10219	// R02 (IN10) W10 RH 작업자위치 이동요구
AND LOAD
OR LOAD
AND NOT   P10230	// R02 (OT33) W10 RH 서보 작업자위치
AND       M0020A	// W10 RH 안전센서 정상
AND NOT   K00051	//  작업자 라인진입 이상
AND       M00241	// W10 RH 로딩 로보트 간섭무
AND       M00242	// W10 RH 언로딩 로보트 간섭무
OUT       M10219	// R02 (IN10) W10 RH 작업자위치 이동요구
; L30
LOAD      M00203	// W10 RH 자동기동
AND       M00279	// W10 RH 1차 작업준비
AND       K00210	// W10 RH 파트 로딩완료
AND       K00211	// W10 RH R02 1차 용접완료
AND       K00217	// W10 RH 언로딩 완료
AND       K00205	// W10 RH 작업완료
AND       M00241	// W10 RH 로딩 로보트 간섭무
AND       M00242	// W10 RH 언로딩 로보트 간섭무
LOAD      M00201	// W10 RH 수동 Mode
LOAD      M0026A	// W10 RH R02 서보 언로딩위치 이동 Pb
OR        M1021A	// R02 (IN11) W10 RH 언로딩위치 이동요구
AND LOAD
OR LOAD
AND NOT   P10231	// R02 (OT34) W10 RH 서보 언로딩위치
AND       M0020A	// W10 RH 안전센서 정상
AND NOT   K00051	//  작업자 라인진입 이상
AND       M00241	// W10 RH 로딩 로보트 간섭무
AND       M00242	// W10 RH 언로딩 로보트 간섭무
AND       F0009A
OUT       M1021A	// R02 (IN11) W10 RH 언로딩위치 이동요구
; L33
LOAD      F0009A
OUT       M1021B	// R02 (IN12)
; L34
LOAD      F0009A
OUT       M1021C	// R02 (IN13)
; L35
LOAD      F0009A
OUT       M1021D	// R02 (IN14)
; L36
LOAD      F0009A
OUT       M1021E	// R02 (IN15)
; L37
LOAD      F0009A
OUT       M1021F	// R02 (IN16)
; L38
LOAD      F0009A
OUT       M10220	// R02 (IN17)

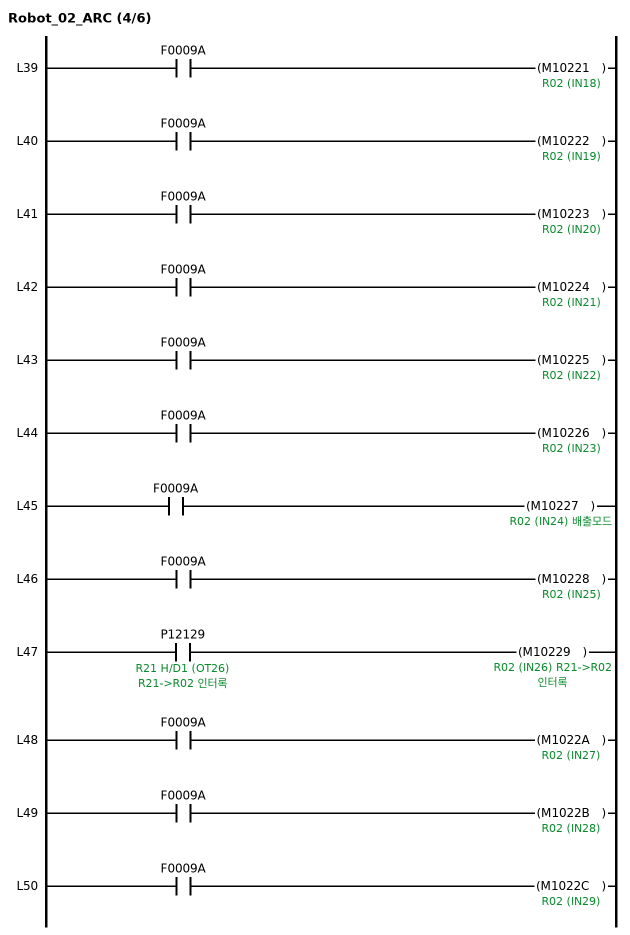
; L39
LOAD      F0009A
OUT       M10221	// R02 (IN18)
; L40
LOAD      F0009A
OUT       M10222	// R02 (IN19)
; L41
LOAD      F0009A
OUT       M10223	// R02 (IN20)
; L42
LOAD      F0009A
OUT       M10224	// R02 (IN21)
; L43
LOAD      F0009A
OUT       M10225	// R02 (IN22)
; L44
LOAD      F0009A
OUT       M10226	// R02 (IN23)
; L45
LOAD      F0009A
OUT       M10227	// R02 (IN24) 배출모드
; L46
LOAD      F0009A
OUT       M10228	// R02 (IN25)
; L47
LOAD      P12129	// R21 H/D1 (OT26) R21->R02 인터록
OUT       M10229	// R02 (IN26) R21->R02 인터록
; L48
LOAD      F0009A
OUT       M1022A	// R02 (IN27)
; L49
LOAD      F0009A
OUT       M1022B	// R02 (IN28)
; L50
LOAD      F0009A
OUT       M1022C	// R02 (IN29)

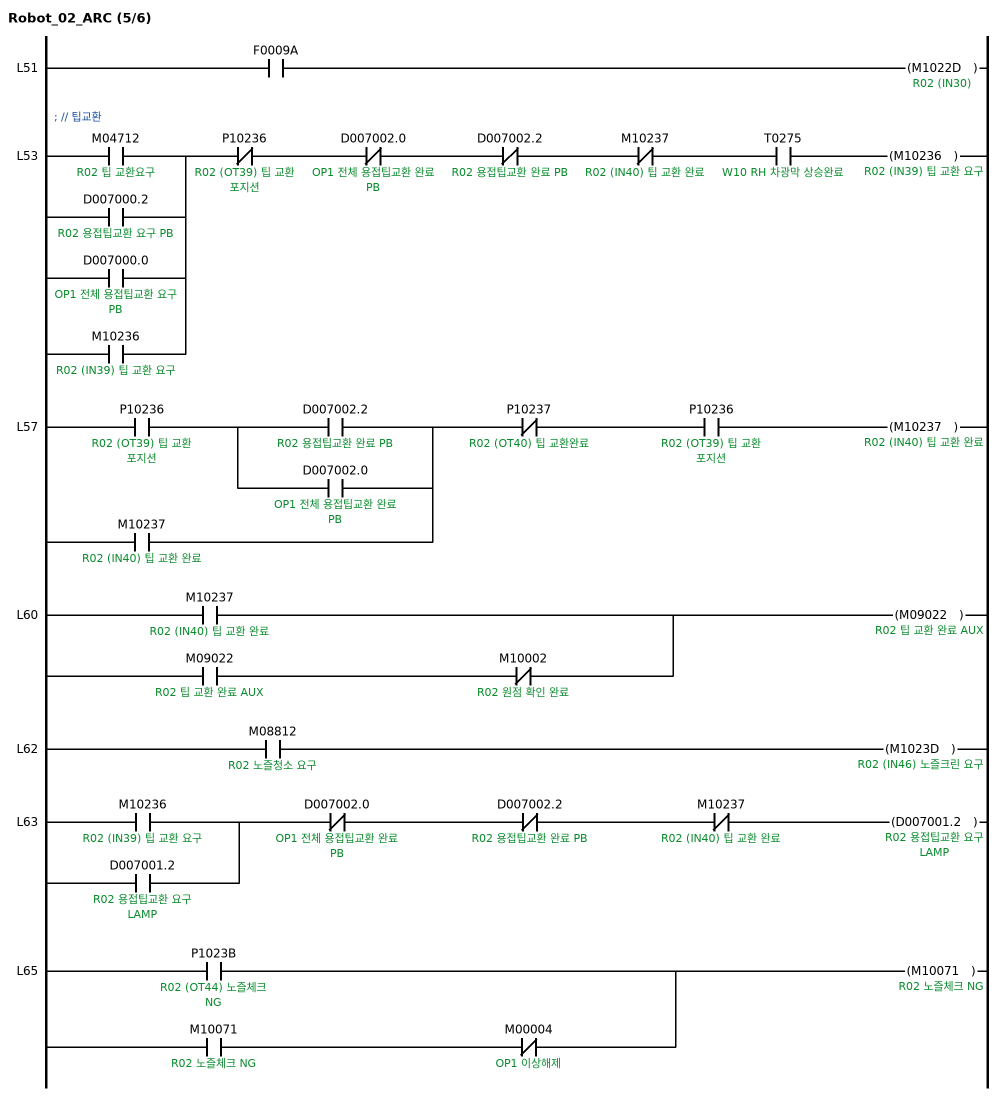
; L51
LOAD      F0009A
OUT       M1022D	// R02 (IN30)
//  // 팁교환
; L53
LOAD      M04712	// R02 팁 교환요구
OR        D007000.2	// R02 용접팁교환 요구 PB
OR        D007000.0	// OP1 전체 용접팁교환 요구 PB
OR        M10236	// R02 (IN39) 팁 교환 요구
AND NOT   P10236	// R02 (OT39) 팁 교환 포지션
AND NOT   D007002.0	// OP1 전체 용접팁교환 완료 PB
AND NOT   D007002.2	// R02 용접팁교환 완료 PB
AND NOT   M10237	// R02 (IN40) 팁 교환 완료
AND       T0275	// W10 RH 차광막 상승완료
OUT       M10236	// R02 (IN39) 팁 교환 요구
; L57
LOAD      P10236	// R02 (OT39) 팁 교환 포지션
LOAD      D007002.2	// R02 용접팁교환 완료 PB
OR        D007002.0	// OP1 전체 용접팁교환 완료 PB
AND LOAD
OR        M10237	// R02 (IN40) 팁 교환 완료
AND NOT   P10237	// R02 (OT40) 팁 교환완료
AND       P10236	// R02 (OT39) 팁 교환 포지션
OUT       M10237	// R02 (IN40) 팁 교환 완료
; L60
LOAD      M10237	// R02 (IN40) 팁 교환 완료
LOAD      M09022	// R02 팁 교환 완료 AUX
AND NOT   M10002	// R02 원점 확인 완료
OR LOAD
OUT       M09022	// R02 팁 교환 완료 AUX
; L62
LOAD      M08812	// R02 노즐청소 요구
OUT       M1023D	// R02 (IN46) 노즐크린 요구
; L63
LOAD      M10236	// R02 (IN39) 팁 교환 요구
OR        D007001.2	// R02 용접팁교환 요구 LAMP
AND NOT   D007002.0	// OP1 전체 용접팁교환 완료 PB
AND NOT   D007002.2	// R02 용접팁교환 완료 PB
AND NOT   M10237	// R02 (IN40) 팁 교환 완료
OUT       D007001.2	// R02 용접팁교환 요구 LAMP
; L65
LOAD      P1023B	// R02 (OT44) 노즐체크 NG
LOAD      M10071	// R02 노즐체크 NG
AND NOT   M00004	// OP1 이상해제
OR LOAD
OUT       M10071	// R02 노즐체크 NG

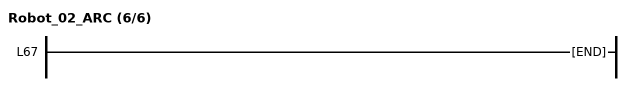
; L67
END

PROGRAM Robot_03_ARC (task: 스캔 프로그램)

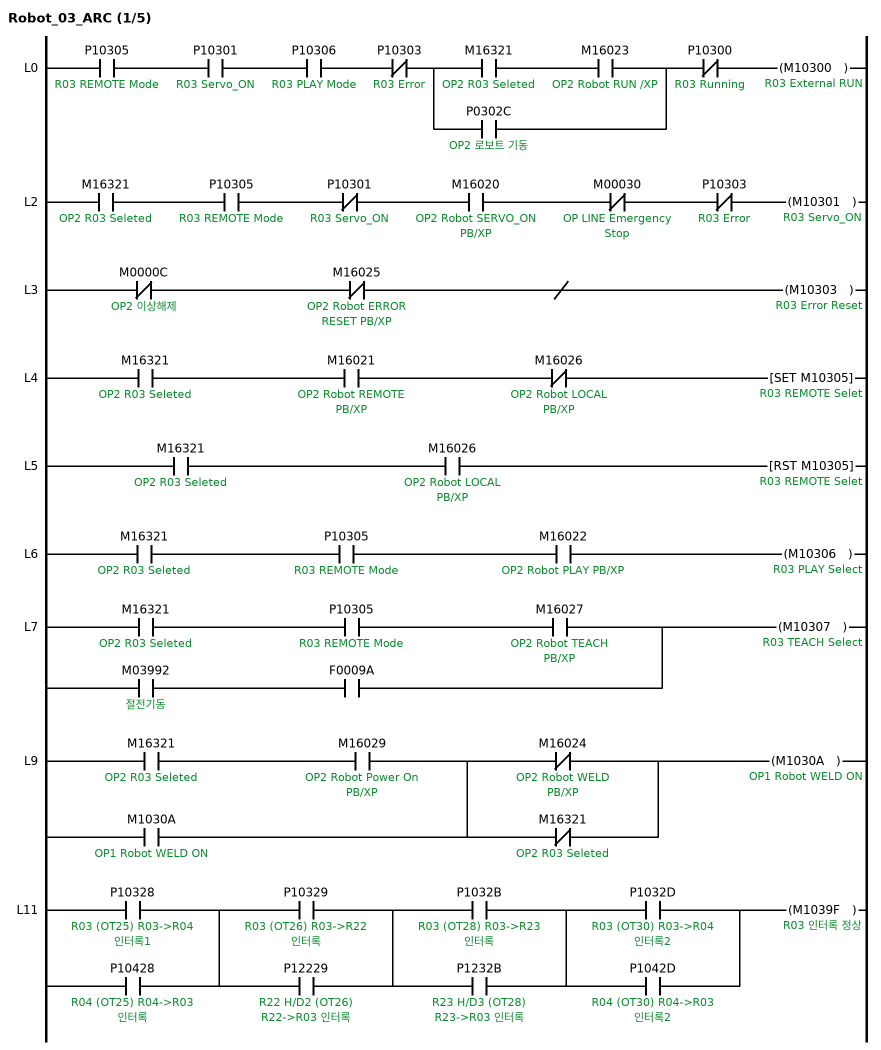
; L0
LOAD      P10305	// R03 REMOTE Mode
AND       P10301	// R03 Servo_ON
AND       P10306	// R03 PLAY Mode
AND NOT   P10303	// R03 Error
LOAD      M16321	// OP2 R03 Seleted
AND       M16023	// OP2 Robot RUN /XP
OR        P0302C	// OP2 로보트 기동
AND LOAD
AND NOT   P10300	// R03 Running
OUT       M10300	// R03 External RUN
; L2
LOAD      M16321	// OP2 R03 Seleted
AND       P10305	// R03 REMOTE Mode
AND NOT   P10301	// R03 Servo_ON
AND       M16020	// OP2 Robot SERVO_ON PB/XP
AND NOT   M00030	// OP LINE Emergency Stop
AND NOT   P10303	// R03 Error
OUT       M10301	// R03 Servo_ON
; L3
LOAD NOT  M0000C	// OP2 이상해제
AND NOT   M16025	// OP2 Robot ERROR RESET PB/XP
NOT
OUT       M10303	// R03 Error Reset
; L4
LOAD      M16321	// OP2 R03 Seleted
AND       M16021	// OP2 Robot REMOTE PB/XP
AND NOT   M16026	// OP2 Robot LOCAL PB/XP
SET       M10305	// R03 REMOTE Selet
; L5
LOAD      M16321	// OP2 R03 Seleted
AND       M16026	// OP2 Robot LOCAL PB/XP
RST       M10305	// R03 REMOTE Selet
; L6
LOAD      M16321	// OP2 R03 Seleted
AND       P10305	// R03 REMOTE Mode
AND       M16022	// OP2 Robot PLAY PB/XP
OUT       M10306	// R03 PLAY Select
; L7
LOAD      M16321	// OP2 R03 Seleted
AND       P10305	// R03 REMOTE Mode
AND       M16027	// OP2 Robot TEACH PB/XP
LOAD      M03992	// 절전기동
AND       F0009A
OR LOAD
OUT       M10307	// R03 TEACH Select
; L9
LOAD      M16321	// OP2 R03 Seleted
AND       M16029	// OP2 Robot Power On PB/XP
OR        M1030A	// OP1 Robot WELD ON
LOAD NOT  M16024	// OP2 Robot WELD PB/XP
OR NOT    M16321	// OP2 R03 Seleted
AND LOAD
OUT       M1030A	// OP1 Robot WELD ON
; L11
LOAD      P10328	// R03 (OT25) R03->R04 인터록1
OR        P10428	// R04 (OT25) R04->R03 인터록
LOAD      P10329	// R03 (OT26) R03->R22 인터록
OR        P12229	// R22 H/D2 (OT26) R22->R03 인터록
AND LOAD
LOAD      P1032B	// R03 (OT28) R03->R23 인터록
OR        P1232B	// R23 H/D3 (OT28) R23->R03 인터록
AND LOAD
LOAD      P1032D	// R03 (OT30) R03->R04 인터록2
OR        P1042D	// R04 (OT30) R04->R03 인터록2
AND LOAD
OUT       M1039F	// R03 인터록 정상

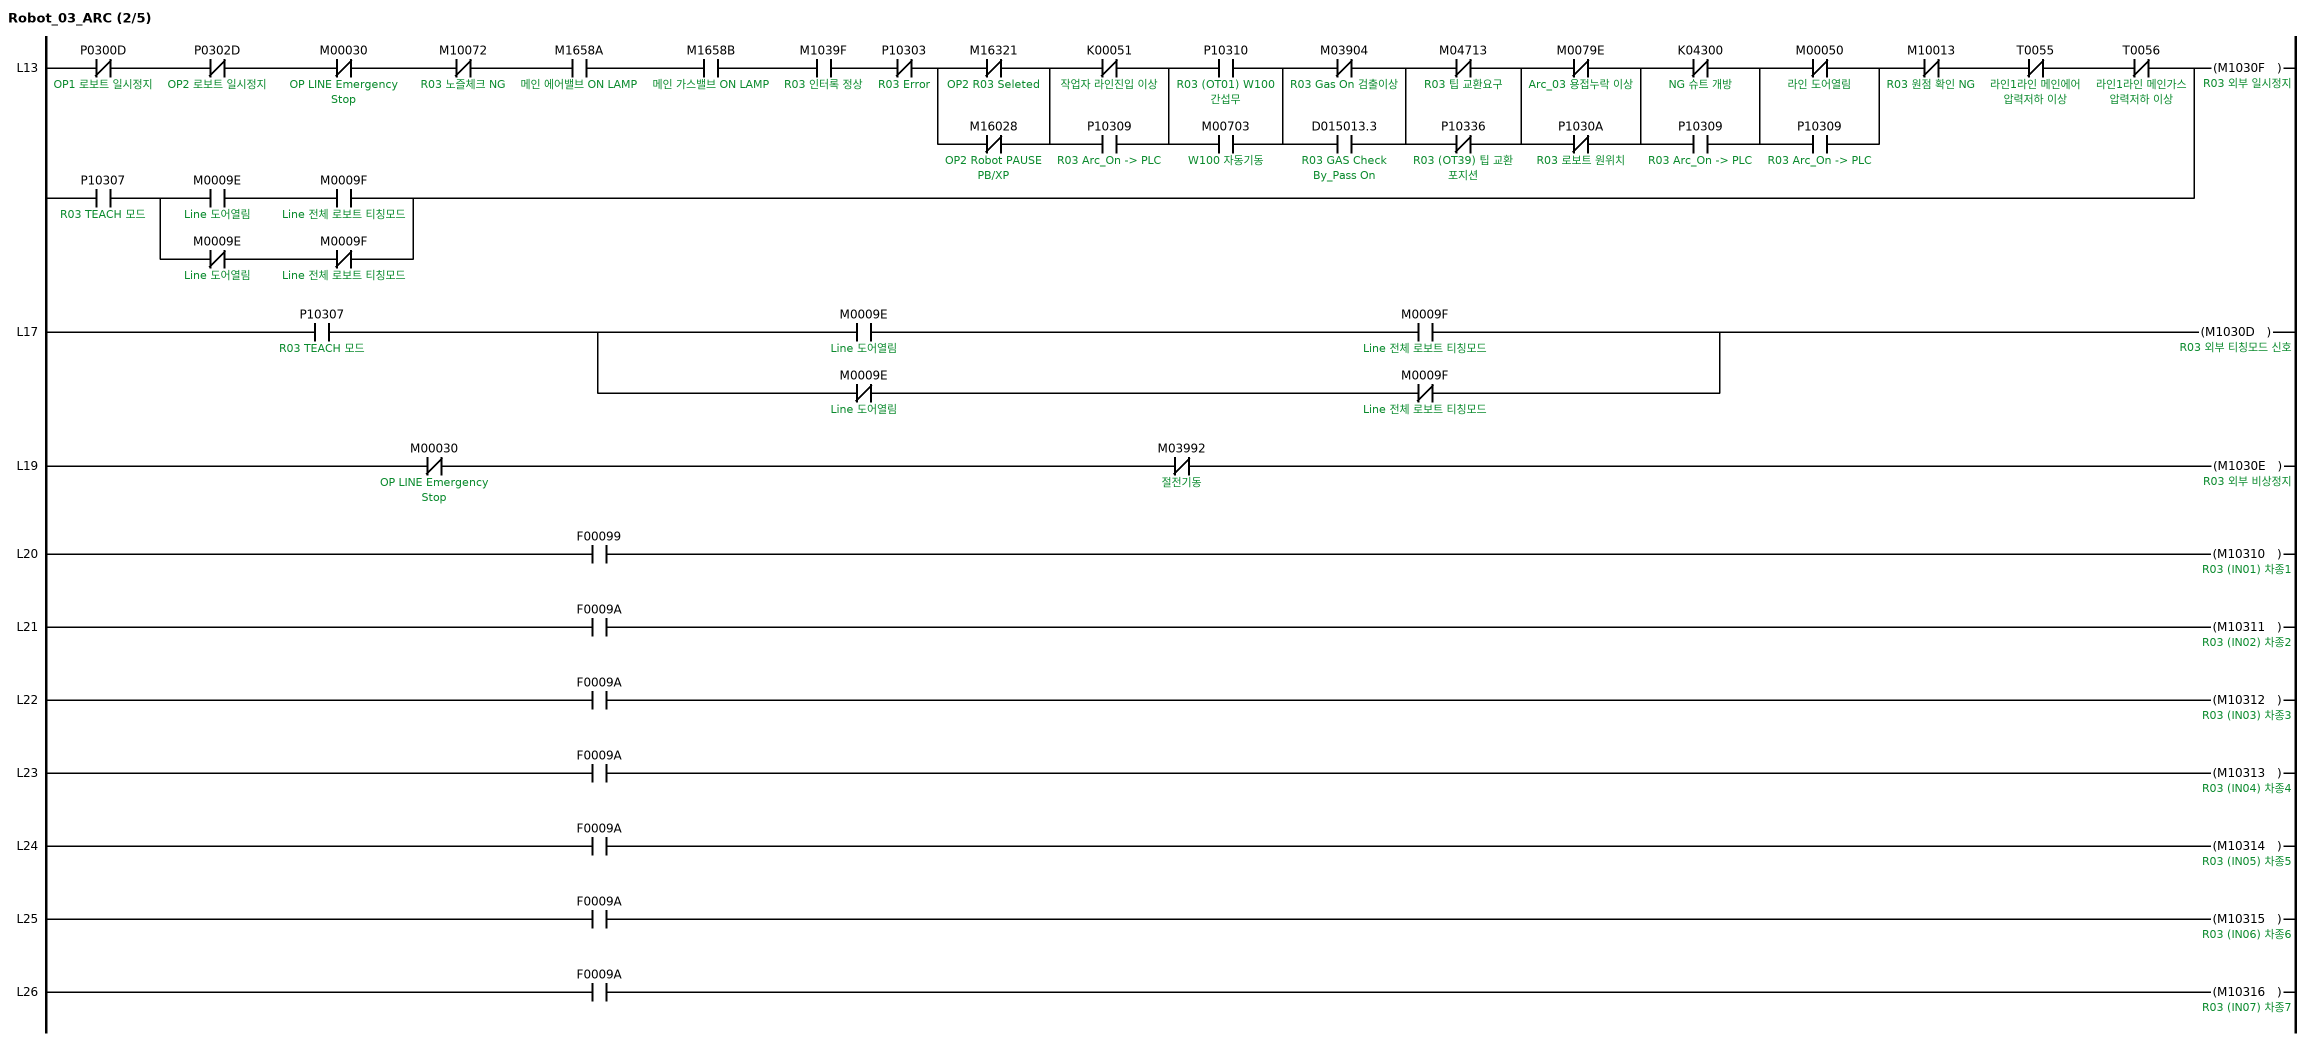
; L13
LOAD NOT  P0300D	// OP1 로보트 일시정지
AND NOT   P0302D	// OP2 로보트 일시정지
AND NOT   M00030	// OP LINE Emergency Stop
AND NOT   M10072	// R03 노즐체크 NG
AND       M1658A	// 메인 에어밸브 ON LAMP
AND       M1658B	// 메인 가스밸브 ON LAMP
AND       M1039F	// R03 인터록 정상
AND NOT   P10303	// R03 Error
LOAD NOT  M16321	// OP2 R03 Seleted
OR NOT    M16028	// OP2 Robot PAUSE PB/XP
AND LOAD
LOAD NOT  K00051	//  작업자 라인진입 이상
OR        P10309	// R03 Arc_On -> PLC
AND LOAD
LOAD      P10310	// R03 (OT01) W100 간섭무
OR        M00703	// W100 자동기동
AND LOAD
LOAD NOT  M03904	// R03 Gas On 검출이상
OR        D015013.3	// R03 GAS Check By_Pass On
AND LOAD
LOAD NOT  M04713	// R03 팁 교환요구
OR NOT    P10336	// R03 (OT39) 팁 교환 포지션
AND LOAD
LOAD NOT  M0079E	// Arc_03 용접누락 이상
OR NOT    P1030A	// R03 로보트 원위치
AND LOAD
LOAD NOT  K04300	// NG 슈트 개방
OR        P10309	// R03 Arc_On -> PLC
AND LOAD
LOAD NOT  M00050	// 라인 도어열림
OR        P10309	// R03 Arc_On -> PLC
AND LOAD
AND NOT   M10013	// R03 원점 확인 NG
AND NOT   T0055	// 라인1라인 메인에어 압력저하 이상
AND NOT   T0056	// 라인1라인 메인가스 압력저하 이상
LOAD      P10307	// R03 TEACH 모드
LOAD      M0009E	// Line 도어열림
AND       M0009F	// Line 전체 로보트 티칭모드
LOAD NOT  M0009E	// Line 도어열림
AND NOT   M0009F	// Line 전체 로보트 티칭모드
OR LOAD
AND LOAD
OR LOAD
OUT       M1030F	// R03 외부 일시정지
; L17
LOAD      P10307	// R03 TEACH 모드
LOAD      M0009E	// Line 도어열림
AND       M0009F	// Line 전체 로보트 티칭모드
LOAD NOT  M0009E	// Line 도어열림
AND NOT   M0009F	// Line 전체 로보트 티칭모드
OR LOAD
AND LOAD
OUT       M1030D	// R03 외부 티칭모드 신호
; L19
LOAD NOT  M00030	// OP LINE Emergency Stop
AND NOT   M03992	// 절전기동
OUT       M1030E	// R03 외부 비상정지 
; L20
LOAD      F00099
OUT       M10310	// R03 (IN01) 차종1
; L21
LOAD      F0009A
OUT       M10311	// R03 (IN02) 차종2
; L22
LOAD      F0009A
OUT       M10312	// R03 (IN03) 차종3
; L23
LOAD      F0009A
OUT       M10313	// R03 (IN04) 차종4
; L24
LOAD      F0009A
OUT       M10314	// R03 (IN05) 차종5
; L25
LOAD      F0009A
OUT       M10315	// R03 (IN06) 차종6
; L26
LOAD      F0009A
OUT       M10316	// R03 (IN07) 차종7

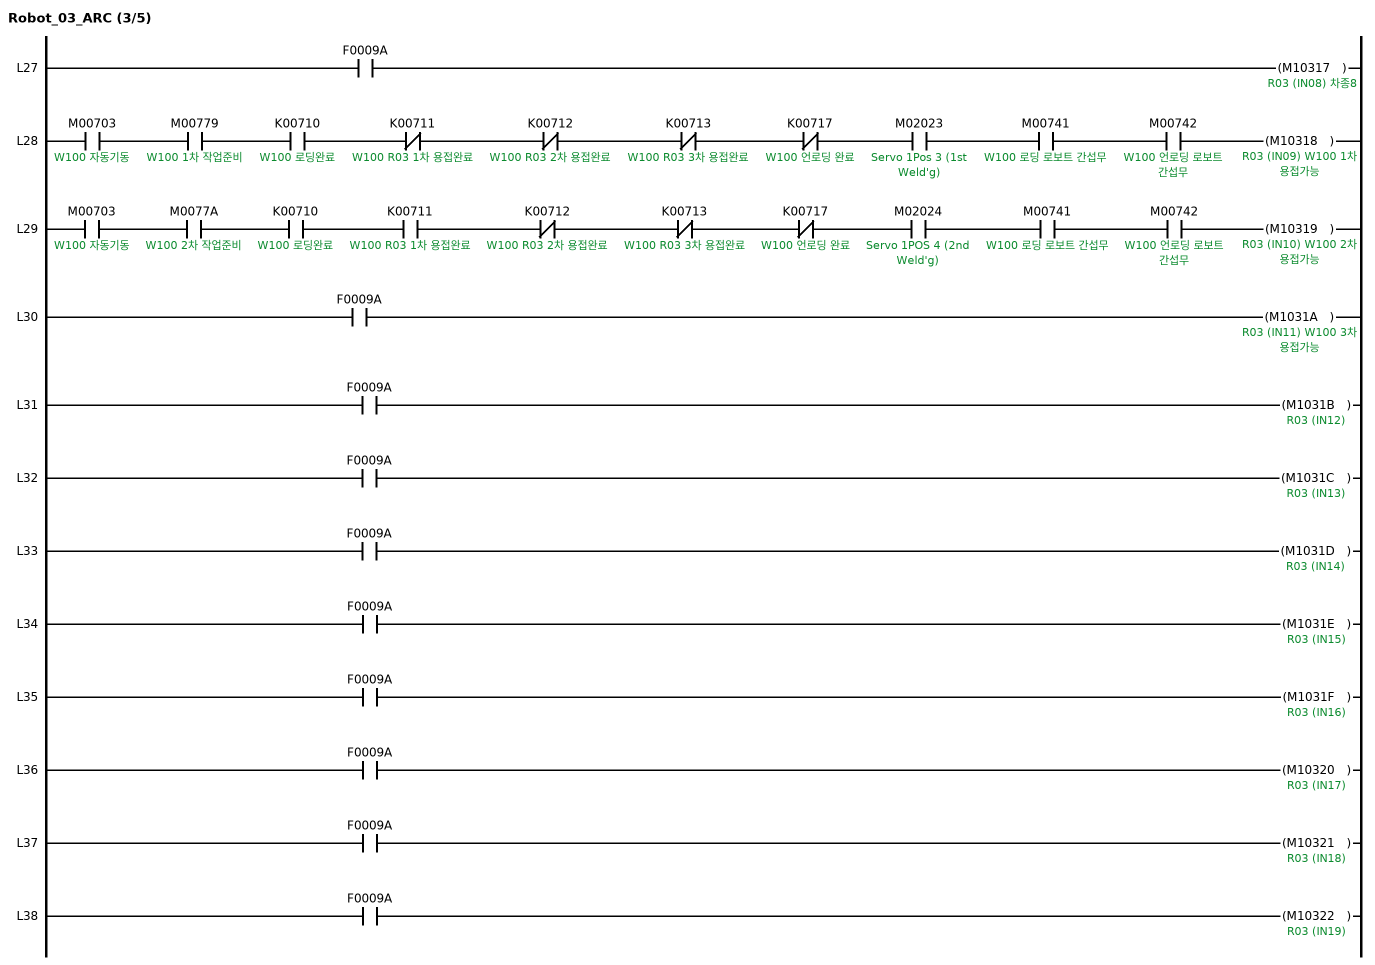
; L27
LOAD      F0009A
OUT       M10317	// R03 (IN08) 차종8
; L28
LOAD      M00703	// W100 자동기동
AND       M00779	// W100 1차 작업준비
AND       K00710	// W100 로딩완료
AND NOT   K00711	// W100 R03 1차 용접완료
AND NOT   K00712	// W100 R03 2차 용접완료
AND NOT   K00713	// W100 R03 3차 용접완료
AND NOT   K00717	// W100 언로딩 완료
AND       M02023	// Servo 1Pos 3 (1st Weld'g)
AND       M00741	// W100 로딩 로보트 간섭무
AND       M00742	// W100 언로딩 로보트 간섭무
OUT       M10318	// R03 (IN09) W100 1차 용접가능
; L29
LOAD      M00703	// W100 자동기동
AND       M0077A	// W100 2차 작업준비
AND       K00710	// W100 로딩완료
AND       K00711	// W100 R03 1차 용접완료
AND NOT   K00712	// W100 R03 2차 용접완료
AND NOT   K00713	// W100 R03 3차 용접완료
AND NOT   K00717	// W100 언로딩 완료
AND       M02024	// Servo 1POS 4 (2nd Weld'g)
AND       M00741	// W100 로딩 로보트 간섭무
AND       M00742	// W100 언로딩 로보트 간섭무
OUT       M10319	// R03 (IN10) W100 2차 용접가능
; L30
LOAD      F0009A
OUT       M1031A	// R03 (IN11) W100 3차 용접가능
; L31
LOAD      F0009A
OUT       M1031B	// R03 (IN12)
; L32
LOAD      F0009A
OUT       M1031C	// R03 (IN13)
; L33
LOAD      F0009A
OUT       M1031D	// R03 (IN14)
; L34
LOAD      F0009A
OUT       M1031E	// R03 (IN15)
; L35
LOAD      F0009A
OUT       M1031F	// R03 (IN16)
; L36
LOAD      F0009A
OUT       M10320	// R03 (IN17)
; L37
LOAD      F0009A
OUT       M10321	// R03 (IN18)
; L38
LOAD      F0009A
OUT       M10322	// R03 (IN19)

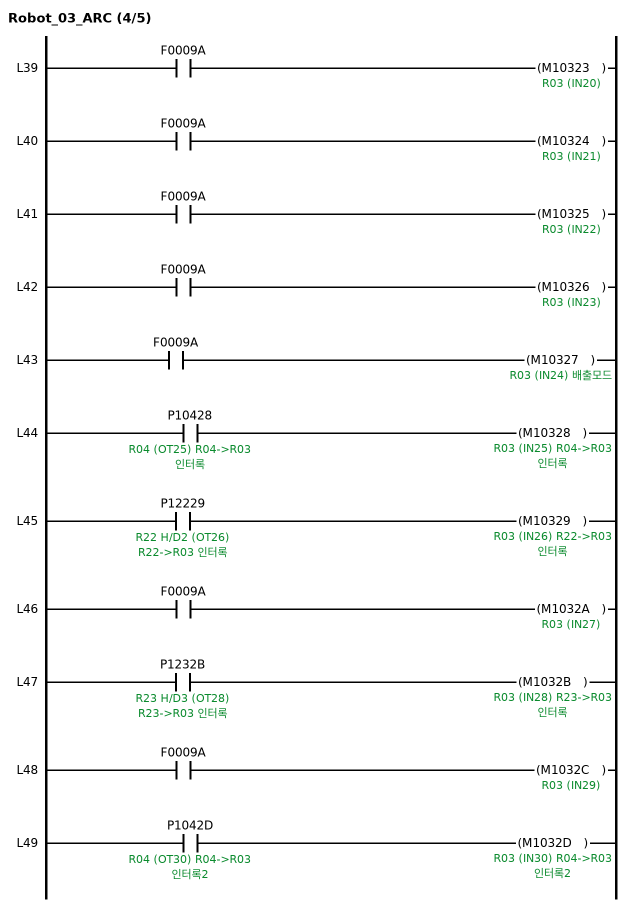
; L39
LOAD      F0009A
OUT       M10323	// R03 (IN20)
; L40
LOAD      F0009A
OUT       M10324	// R03 (IN21)
; L41
LOAD      F0009A
OUT       M10325	// R03 (IN22)
; L42
LOAD      F0009A
OUT       M10326	// R03 (IN23)
; L43
LOAD      F0009A
OUT       M10327	// R03 (IN24) 배출모드
; L44
LOAD      P10428	// R04 (OT25) R04->R03 인터록
OUT       M10328	// R03 (IN25) R04->R03 인터록
; L45
LOAD      P12229	// R22 H/D2 (OT26) R22->R03 인터록
OUT       M10329	// R03 (IN26) R22->R03 인터록
; L46
LOAD      F0009A
OUT       M1032A	// R03 (IN27)
; L47
LOAD      P1232B	// R23 H/D3 (OT28) R23->R03 인터록
OUT       M1032B	// R03 (IN28) R23->R03 인터록
; L48
LOAD      F0009A
OUT       M1032C	// R03 (IN29)
; L49
LOAD      P1042D	// R04 (OT30) R04->R03 인터록2
OUT       M1032D	// R03 (IN30) R04->R03 인터록2

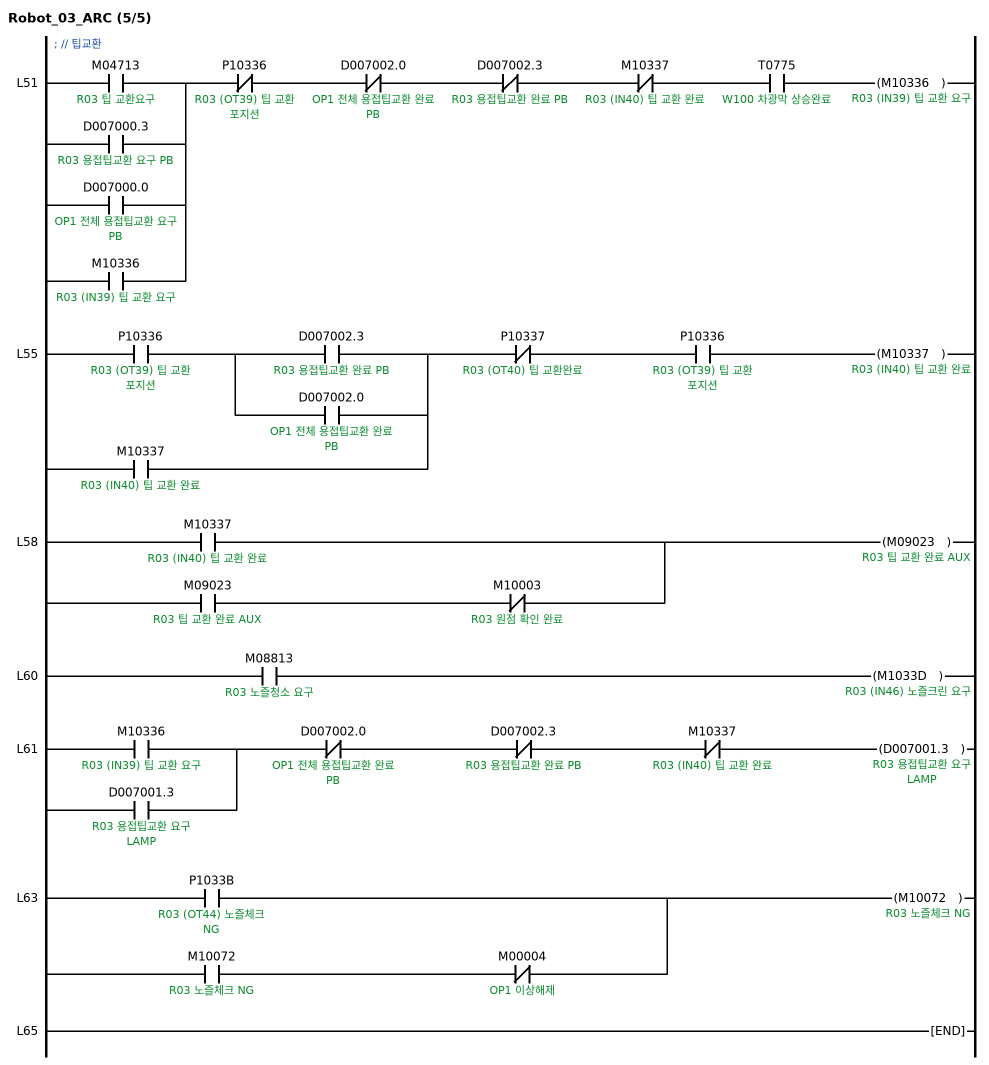
//  // 팁교환
; L51
LOAD      M04713	// R03 팁 교환요구
OR        D007000.3	// R03 용접팁교환 요구 PB
OR        D007000.0	// OP1 전체 용접팁교환 요구 PB
OR        M10336	// R03 (IN39) 팁 교환 요구
AND NOT   P10336	// R03 (OT39) 팁 교환 포지션
AND NOT   D007002.0	// OP1 전체 용접팁교환 완료 PB
AND NOT   D007002.3	// R03 용접팁교환 완료 PB
AND NOT   M10337	// R03 (IN40) 팁 교환 완료
AND       T0775	// W100 차광막 상승완료
OUT       M10336	// R03 (IN39) 팁 교환 요구
; L55
LOAD      P10336	// R03 (OT39) 팁 교환 포지션
LOAD      D007002.3	// R03 용접팁교환 완료 PB
OR        D007002.0	// OP1 전체 용접팁교환 완료 PB
AND LOAD
OR        M10337	// R03 (IN40) 팁 교환 완료
AND NOT   P10337	// R03 (OT40) 팁 교환완료
AND       P10336	// R03 (OT39) 팁 교환 포지션
OUT       M10337	// R03 (IN40) 팁 교환 완료
; L58
LOAD      M10337	// R03 (IN40) 팁 교환 완료
LOAD      M09023	// R03 팁 교환 완료 AUX
AND NOT   M10003	// R03 원점 확인 완료
OR LOAD
OUT       M09023	// R03 팁 교환 완료 AUX
; L60
LOAD      M08813	// R03 노즐청소 요구
OUT       M1033D	// R03 (IN46) 노즐크린 요구
; L61
LOAD      M10336	// R03 (IN39) 팁 교환 요구
OR        D007001.3	// R03 용접팁교환 요구 LAMP
AND NOT   D007002.0	// OP1 전체 용접팁교환 완료 PB
AND NOT   D007002.3	// R03 용접팁교환 완료 PB
AND NOT   M10337	// R03 (IN40) 팁 교환 완료
OUT       D007001.3	// R03 용접팁교환 요구 LAMP
; L63
LOAD      P1033B	// R03 (OT44) 노즐체크 NG
LOAD      M10072	// R03 노즐체크 NG
AND NOT   M00004	// OP1 이상해제
OR LOAD
OUT       M10072	// R03 노즐체크 NG
; L65
END

PROGRAM Robot_04_ARC (task: 스캔 프로그램)

